LIN {X 0,Y 98.445,Z 539.877,A -85,B 0,C 180,E1 -26554.094,E2 -26554.094} C_VEL
LIN {X 0,Y 100.057,Z 537.535,A -85,B 0,C 180,E1 -26562.164,E2 -26562.164} C_VEL
LIN {X 0,Y 102.288,Z 534.743,A -85,B 0,C 180,E1 -26568.01,E2 -26568.01} C_VEL
LIN {X 0,Y 105.398,Z 531.036,A -85,B 0,C 180,E1 -26573.583,E2 -26573.583} C_VEL
LIN {X 0,Y 109.416,Z 526.315,A -85,B 0,C 180,E1 -26578.798,E2 -26578.798} C_VEL
LIN {X 0,Y 115.169,Z 519.342,A -85,B 0,C 180,E1 -26584.364,E2 -26584.364} C_VEL
LIN {X 0,Y 120.723,Z 511.905,A -85,B 0,C 180,E1 -26588.741,E2 -26588.741} C_VEL
LIN {X 0,Y 127.011,Z 502.792,A -85,B 0,C 180,E1 -26592.674,E2 -26592.674} C_VEL
LIN {X 0,Y 132.642,Z 493.502,A -85,B 0,C 180,E1 -26595.666,E2 -26595.666} C_VEL
LIN {X 0,Y 137.859,Z 483.367,A -85,B 0,C 180,E1 -26598.207,E2 -26598.207} C_VEL
LIN {X 0,Y 142.816,Z 472.376,A -85,B 0,C 180,E1 -26600.227,E2 -26600.227} C_VEL
LIN {X 0,Y 147.276,Z 460.103,A -85,B 0,C 180,E1 -26601.94,E2 -26601.94} C_VEL
LIN {X 0,Y 151.028,Z 446.667,A -85,B 0,C 180,E1 -26603.297,E2 -26603.297} C_VEL
LIN {X 0,Y 153.636,Z 433.846,A -85,B 0,C 180,E1 -26604.14,E2 -26604.14} C_VEL
LIN {X 0,Y 155.312,Z 419.503,A -85,B 0,C 180,E1 -26604.738,E2 -26604.738} C_VEL
LIN {X 0,Y 158.37,Z 382.753,A -85,B 0,C 180,E1 -26606.002,E2 -26606.002} C_VEL
LIN {X 0,Y 155.054,Z 373.648,A -85,B 0,C 180,E1 -26608.871,E2 -26608.871} C_VEL
LIN {X 0,Y 151.004,Z 364.193,A -85,B 0,C 180,E1 -26612.816,E2 -26612.816} C_VEL
LIN {X 0,Y 148.386,Z 358.823,A -85,B 0,C 180,E1 -26615.763,E2 -26615.763} C_VEL
LIN {X 0,Y 146.643,Z 355.474,A -85,B 0,C 180,E1 -26617.992,E2 -26617.992} C_VEL
LIN {X 0,Y 144.423,Z 351.265,A -85,B 0,C 180,E1 -26621.329,E2 -26621.329} C_VEL
LIN {X 0,Y 141.659,Z 346.333,A -85,B 0,C 180,E1 -26626.943,E2 -26626.943} C_VEL
LIN {X 0,Y 139.867,Z 343.216,A -85,B 0,C 180,E1 -26633.833,E2 -26633.833} C_VEL
LIN {X 0,Y 139.693,Z 342.139,A -85,B 0,C 180,E1 -26638.558,E2 -26638.558} C_VEL
LIN {X 0,Y 139.869,Z 342.535,A -85,B 0,C 180,E1 -26641.079,E2 -26641.079} C_VEL
LIN {X 0,Y 141.875,Z 345.546,A -85,B 0,C 180,E1 -26648.747,E2 -26648.747} C_VEL
LIN {X 0,Y 145.014,Z 350.889,A -85,B 0,C 180,E1 -26654.829,E2 -26654.829} C_VEL
LIN {X 0,Y 147.601,Z 355.381,A -85,B 0,C 180,E1 -26658.449,E2 -26658.449} C_VEL
LIN {X 0,Y 150.224,Z 360.312,A -85,B 0,C 180,E1 -26661.527,E2 -26661.527} C_VEL
LIN {X 0,Y 153.271,Z 366.548,A -85,B 0,C 180,E1 -26664.643,E2 -26664.643} C_VEL
LIN {X 0,Y 156.605,Z 374.178,A -85,B 0,C 180,E1 -26667.662,E2 -26667.662} C_VEL
LIN {X 0,Y 158.852,Z 380.327,A -85,B 0,C 180,E1 -26669.571,E2 -26669.571} C_VEL
LIN {X 0,Y 154.248,Z 429.807,A -85,B 0,C 180,E1 -26671.258,E2 -26671.258} C_VEL
LIN {X 0,Y 151.821,Z 443.678,A -85,B 0,C 180,E1 -26672.049,E2 -26672.049} C_VEL
LIN {X 0,Y 148.088,Z 457.884,A -85,B 0,C 180,E1 -26673.235,E2 -26673.235} C_VEL
LIN {X 0,Y 144.21,Z 469.529,A -85,B 0,C 180,E1 -26674.676,E2 -26674.676} C_VEL
LIN {X 0,Y 139.076,Z 481.819,A -85,B 0,C 180,E1 -26676.659,E2 -26676.659} C_VEL
LIN {X 0,Y 133.918,Z 492.462,A -85,B 0,C 180,E1 -26679.031,E2 -26679.031} C_VEL
LIN {X 0,Y 127.84,Z 503.024,A -85,B 0,C 180,E1 -26682.085,E2 -26682.085} C_VEL
LIN {X 0,Y 121.244,Z 512.968,A -85,B 0,C 180,E1 -26685.927,E2 -26685.927} C_VEL
LIN {X 0,Y 115.415,Z 521.126,A -85,B 0,C 180,E1 -26690.256,E2 -26690.256} C_VEL
LIN {X 0,Y 110.286,Z 527.828,A -85,B 0,C 180,E1 -26695.004,E2 -26695.004} C_VEL
LIN {X 0,Y 106.098,Z 533.312,A -85,B 0,C 180,E1 -26700.212,E2 -26700.212} C_VEL
LIN {X 0,Y 102.683,Z 537.722,A -85,B 0,C 180,E1 -26705.754,E2 -26705.754} C_VEL
LIN {X 0,Y 99.505,Z 542.086,A -85,B 0,C 180,E1 -26713.59,E2 -26713.59} C_VEL
LIN {X 0,Y 98.09,Z 544.903,A -85,B 0,C 180,E1 -26721.762,E2 -26721.762} C_VEL
LIN {X 0,Y 97.925,Z 545.745,A -85,B 0,C 180,E1 -26725.885,E2 -26725.885} C_VEL
LIN {X 0,Y 98.071,Z 546.205,A -85,B 0,C 180,E1 -26730,E2 -26730} C_VEL
LIN {X 0,Y 97.935,Z 546.283,A -85,B 0,C 180,E1 -26734.115,E2 -26734.115} C_VEL
LIN {X 0,Y 98.656,Z 545.36,A -85,B 0,C 180,E1 -26742.34,E2 -26742.34} C_VEL
LIN {X 0,Y 100.917,Z 542.994,A -85,B 0,C 180,E1 -26750.377,E2 -26750.377} C_VEL
LIN {X 0,Y 103.898,Z 540.216,A -85,B 0,C 180,E1 -26756.083,E2 -26756.083} C_VEL
LIN {X 0,Y 108.683,Z 535.456,A -85,B 0,C 180,E1 -26762.793,E2 -26762.793} C_VEL
LIN {X 0,Y 113.953,Z 530.064,A -85,B 0,C 180,E1 -26768.078,E2 -26768.078} C_VEL
LIN {X 0,Y 120.709,Z 522.772,A -85,B 0,C 180,E1 -26773.165,E2 -26773.165} C_VEL
LIN {X 0,Y 127.182,Z 515.033,A -85,B 0,C 180,E1 -26777.069,E2 -26777.069} C_VEL
LIN {X 0,Y 134.163,Z 505.579,A -85,B 0,C 180,E1 -26780.593,E2 -26780.593} C_VEL
LIN {X 0,Y 138.497,Z 498.922,A -85,B 0,C 180,E1 -26782.545,E2 -26782.545} C_VEL
LIN {X 0,Y 140.818,Z 494.528,A -85,B 0,C 180,E1 -26783.862,E2 -26783.862} C_VEL
LIN {X 0,Y 143.313,Z 487.207,A -85,B 0,C 180,E1 -26786.378,E2 -26786.378} C_VEL
LIN {X 0,Y 145.665,Z 479.481,A -85,B 0,C 180,E1 -26788.651,E2 -26788.651} C_VEL
LIN {X 0,Y 147.649,Z 474.457,A -85,B 0,C 180,E1 -26789.573,E2 -26789.573} C_VEL
LIN {X 0,Y 151.923,Z 464.012,A -85,B 0,C 180,E1 -26790.827,E2 -26790.827} C_VEL
LIN {X 0,Y 156.228,Z 450.743,A -85,B 0,C 180,E1 -26791.985,E2 -26791.985} C_VEL
LIN {X 0,Y 159.545,Z 436.77,A -85,B 0,C 180,E1 -26792.801,E2 -26792.801} C_VEL
LIN {X 0,Y 161.561,Z 422.766,A -85,B 0,C 180,E1 -26793.348,E2 -26793.348} C_VEL
LIN {X 0,Y 164.54,Z 391.448,A -85,B 0,C 180,E1 -26794.328,E2 -26794.328} C_VEL
LIN {X 0,Y 161.223,Z 382.87,A -85,B 0,C 180,E1 -26797.832,E2 -26797.832} C_VEL
LIN {X 0,Y 158.331,Z 376.36,A -85,B 0,C 180,E1 -26801.396,E2 -26801.396} C_VEL
LIN {X 0,Y 156.515,Z 372.65,A -85,B 0,C 180,E1 -26804.041,E2 -26804.041} C_VEL
LIN {X 0,Y 154.7,Z 369.18,A -85,B 0,C 180,E1 -26807.205,E2 -26807.205} C_VEL
LIN {X 0,Y 152.882,Z 365.51,A -85,B 0,C 180,E1 -26811.596,E2 -26811.596} C_VEL
LIN {X 0,Y 151.763,Z 363.688,A -85,B 0,C 180,E1 -26816.018,E2 -26816.018} C_VEL
LIN {X 0,Y 151.454,Z 362.725,A -85,B 0,C 180,E1 -26820.001,E2 -26820.001} C_VEL
LIN {X 0,Y 151.968,Z 364.564,A -85,B 0,C 180,E1 -26825.974,E2 -26825.974} C_VEL
LIN {X 0,Y 153.384,Z 367.616,A -85,B 0,C 180,E1 -26830.729,E2 -26830.729} C_VEL
LIN {X 0,Y 155.623,Z 372.465,A -85,B 0,C 180,E1 -26835.387,E2 -26835.387} C_VEL
LIN {X 0,Y 157.722,Z 377.127,A -85,B 0,C 180,E1 -26838.663,E2 -26838.663} C_VEL
LIN {X 0,Y 160.038,Z 382.681,A -85,B 0,C 180,E1 -26841.683,E2 -26841.683} C_VEL
LIN {X 0,Y 163.374,Z 391.759,A -85,B 0,C 180,E1 -26845.411,E2 -26845.411} C_VEL
LIN {X 0,Y 164.211,Z 394.346,A -85,B 0,C 180,E1 -26846.277,E2 -26846.277} C_VEL
LIN {X 0,Y 160.771,Z 429.208,A -85,B 0,C 180,E1 -26847.356,E2 -26847.356} C_VEL
LIN {X 0,Y 158.038,Z 443.429,A -85,B 0,C 180,E1 -26848.062,E2 -26848.062} C_VEL
LIN {X 0,Y 154.281,Z 456.733,A -85,B 0,C 180,E1 -26849.069,E2 -26849.069} C_VEL
LIN {X 0,Y 149.779,Z 468.983,A -85,B 0,C 180,E1 -26850.437,E2 -26850.437} C_VEL
LIN {X 0,Y 144.308,Z 480.728,A -85,B 0,C 180,E1 -26852.202,E2 -26852.202} C_VEL
LIN {X 0,Y 138.053,Z 491.906,A -85,B 0,C 180,E1 -26854.496,E2 -26854.496} C_VEL
LIN {X 0,Y 131.861,Z 501.111,A -85,B 0,C 180,E1 -26856.921,E2 -26856.921} C_VEL
LIN {X 0,Y 124.436,Z 510.659,A -85,B 0,C 180,E1 -26860.319,E2 -26860.319} C_VEL
LIN {X 0,Y 117.571,Z 518.415,A -85,B 0,C 180,E1 -26864.167,E2 -26864.167} C_VEL
LIN {X 0,Y 111.241,Z 524.729,A -85,B 0,C 180,E1 -26868.443,E2 -26868.443} C_VEL
LIN {X 0,Y 105.741,Z 529.827,A -85,B 0,C 180,E1 -26873.261,E2 -26873.261} C_VEL
LIN {X 0,Y 100.987,Z 533.857,A -85,B 0,C 180,E1 -26878.537,E2 -26878.537} C_VEL
LIN {X 0,Y 96.967,Z 536.935,A -85,B 0,C 180,E1 -26884.223,E2 -26884.223} C_VEL
LIN {X 0,Y 93.331,Z 539.678,A -85,B 0,C 180,E1 -26892.47,E2 -26892.47} C_VEL
LIN {X 0,Y 91.373,Z 540.926,A -85,B 0,C 180,E1 -26901.151,E2 -26901.151} C_VEL
LIN {X 0,Y 91.052,Z 540.719,A -85,B 0,C 180,E1 -26910,E2 -26910} C_VEL
LIN {X 0,Y 91.387,Z 540.09,A -85,B 0,C 180,E1 -26914.41,E2 -26914.41} C_VEL
LIN {X 0,Y 93.142,Z 537.76,A -85,B 0,C 180,E1 -26923.083,E2 -26923.083} C_VEL
LIN {X 0,Y 95.566,Z 534.981,A -85,B 0,C 180,E1 -26929.325,E2 -26929.325} C_VEL
LIN {X 0,Y 98.954,Z 531.289,A -85,B 0,C 180,E1 -26935.222,E2 -26935.222} C_VEL
LIN {X 0,Y 103.263,Z 526.585,A -85,B 0,C 180,E1 -26940.693,E2 -26940.693} C_VEL
LIN {X 0,Y 109.397,Z 519.632,A -85,B 0,C 180,E1 -26946.458,E2 -26946.458} C_VEL
LIN {X 0,Y 115.273,Z 512.221,A -85,B 0,C 180,E1 -26950.95,E2 -26950.95} C_VEL
LIN {X 0,Y 121.91,Z 503.144,A -85,B 0,C 180,E1 -26954.926,E2 -26954.926} C_VEL
LIN {X 0,Y 126.607,Z 495.855,A -85,B 0,C 180,E1 -26957.349,E2 -26957.349} C_VEL
LIN {X 0,Y 132.616,Z 485.046,A -85,B 0,C 180,E1 -26960.211,E2 -26960.211} C_VEL
LIN {X 0,Y 138.024,Z 473.823,A -85,B 0,C 180,E1 -26962.335,E2 -26962.335} C_VEL
LIN {X 0,Y 142.375,Z 462.739,A -85,B 0,C 180,E1 -26963.93,E2 -26963.93} C_VEL
LIN {X 0,Y 146.275,Z 449.923,A -85,B 0,C 180,E1 -26965.307,E2 -26965.307} C_VEL
LIN {X 0,Y 149.398,Z 436.136,A -85,B 0,C 180,E1 -26966.274,E2 -26966.274} C_VEL
LIN {X 0,Y 151.259,Z 422.842,A -85,B 0,C 180,E1 -26966.869,E2 -26966.869} C_VEL
LIN {X 0,Y 154.537,Z 385.412,A -85,B 0,C 180,E1 -26968.135,E2 -26968.135} C_VEL
LIN {X 0,Y 151.217,Z 376.194,A -85,B 0,C 180,E1 -26971.37,E2 -26971.37} C_VEL
LIN {X 0,Y 147.848,Z 368.107,A -85,B 0,C 180,E1 -26975.115,E2 -26975.115} C_VEL
LIN {X 0,Y 145.186,Z 362.309,A -85,B 0,C 180,E1 -26978.625,E2 -26978.625} C_VEL
LIN {X 0,Y 142.907,Z 357.801,A -85,B 0,C 180,E1 -26982.283,E2 -26982.283} C_VEL
LIN {X 0,Y 140.493,Z 353.11,A -85,B 0,C 180,E1 -26987.651,E2 -26987.651} C_VEL
LIN {X 0,Y 138.91,Z 350.107,A -85,B 0,C 180,E1 -26994.566,E2 -26994.566} C_VEL
LIN {X 0,Y 138.826,Z 349.201,A -85,B 0,C 180,E1 -26998.549,E2 -26998.549} C_VEL
LIN {X 0,Y 138.996,Z 349.636,A -85,B 0,C 180,E1 -27001.085,E2 -27001.085} C_VEL
LIN {X 0,Y 140.772,Z 352.508,A -85,B 0,C 180,E1 -27008.251,E2 -27008.251} C_VEL
LIN {X 0,Y 143.481,Z 357.418,A -85,B 0,C 180,E1 -27013.904,E2 -27013.904} C_VEL
LIN {X 0,Y 145.753,Z 361.641,A -85,B 0,C 180,E1 -27017.358,E2 -27017.358} C_VEL
LIN {X 0,Y 148.347,Z 366.881,A -85,B 0,C 180,E1 -27020.653,E2 -27020.653} C_VEL
LIN {X 0,Y 151.329,Z 373.477,A -85,B 0,C 180,E1 -27023.908,E2 -27023.908} C_VEL
LIN {X 0,Y 154.651,Z 381.947,A -85,B 0,C 180,E1 -27027.119,E2 -27027.119} C_VEL
LIN {X 0,Y 154.977,Z 382.874,A -85,B 0,C 180,E1 -27027.419,E2 -27027.419} C_VEL
LIN {X 0,Y 150.424,Z 430.008,A -85,B 0,C 180,E1 -27029.013,E2 -27029.013} C_VEL
LIN {X 0,Y 147.841,Z 444.116,A -85,B 0,C 180,E1 -27029.807,E2 -27029.807} C_VEL
LIN {X 0,Y 144.302,Z 457.156,A -85,B 0,C 180,E1 -27030.865,E2 -27030.865} C_VEL
LIN {X 0,Y 140.279,Z 468.942,A -85,B 0,C 180,E1 -27032.283,E2 -27032.283} C_VEL
LIN {X 0,Y 134.925,Z 481.329,A -85,B 0,C 180,E1 -27034.22,E2 -27034.22} C_VEL
LIN {X 0,Y 128.968,Z 493.038,A -85,B 0,C 180,E1 -27036.828,E2 -27036.828} C_VEL
LIN {X 0,Y 123.148,Z 502.661,A -85,B 0,C 180,E1 -27039.608,E2 -27039.608} C_VEL
LIN {X 0,Y 116.234,Z 512.64,A -85,B 0,C 180,E1 -27043.485,E2 -27043.485} C_VEL
LIN {X 0,Y 110.002,Z 520.823,A -85,B 0,C 180,E1 -27047.869,E2 -27047.869} C_VEL
LIN {X 0,Y 104.503,Z 527.547,A -85,B 0,C 180,E1 -27052.753,E2 -27052.753} C_VEL
LIN {X 0,Y 99.89,Z 533.093,A -85,B 0,C 180,E1 -27058.217,E2 -27058.217} C_VEL
LIN {X 0,Y 95.158,Z 538.74,A -85,B 0,C 180,E1 -27066.034,E2 -27066.034} C_VEL
LIN {X 0,Y 92.674,Z 541.853,A -85,B 0,C 180,E1 -27072.342,E2 -27072.342} C_VEL
LIN {X 0,Y 91.056,Z 544.683,A -85,B 0,C 180,E1 -27081.12,E2 -27081.12} C_VEL
LIN {X 0,Y 90.824,Z 545.535,A -85,B 0,C 180,E1 -27085.562,E2 -27085.562} C_VEL
LIN {X 0,Y 90.969,Z 546.003,A -85,B 0,C 180,E1 -27090,E2 -27090} C_VEL
LIN {X 0,Y 90.861,Z 546.087,A -85,B 0,C 180,E1 -27094.436,E2 -27094.436} C_VEL
LIN {X 0,Y 91.684,Z 545.173,A -85,B 0,C 180,E1 -27103.295,E2 -27103.295} C_VEL
LIN {X 0,Y 94.253,Z 542.817,A -85,B 0,C 180,E1 -27111.89,E2 -27111.89} C_VEL
LIN {X 0,Y 97.518,Z 540.049,A -85,B 0,C 180,E1 -27117.933,E2 -27117.933} C_VEL
LIN {X 0,Y 102.319,Z 535.68,A -85,B 0,C 180,E1 -27124.49,E2 -27124.49} C_VEL
LIN {X 0,Y 108.424,Z 529.917,A -85,B 0,C 180,E1 -27130.405,E2 -27130.405} C_VEL
LIN {X 0,Y 115.578,Z 522.633,A -85,B 0,C 180,E1 -27135.6,E2 -27135.6} C_VEL
LIN {X 0,Y 122.433,Z 514.904,A -85,B 0,C 180,E1 -27139.515,E2 -27139.515} C_VEL
LIN {X 0,Y 129.75,Z 505.459,A -85,B 0,C 180,E1 -27143.028,E2 -27143.028} C_VEL
LIN {X 0,Y 136.785,Z 494.847,A -85,B 0,C 180,E1 -27145.944,E2 -27145.944} C_VEL
LIN {X 0,Y 143.528,Z 482.98,A -85,B 0,C 180,E1 -27148.296,E2 -27148.296} C_VEL
LIN {X 0,Y 147.649,Z 474.457,A -85,B 0,C 180,E1 -27149.573,E2 -27149.573} C_VEL
LIN {X 0,Y 149.552,Z 469.346,A -85,B 0,C 180,E1 -27150.423,E2 -27150.423} C_VEL
LIN {X 0,Y 151.378,Z 460.868,A -85,B 0,C 180,E1 -27152.289,E2 -27152.289} C_VEL
LIN {X 0,Y 152.891,Z 452.178,A -85,B 0,C 180,E1 -27153.992,E2 -27153.992} C_VEL
LIN {X 0,Y 154.136,Z 446.643,A -85,B 0,C 180,E1 -27154.595,E2 -27154.595} C_VEL
LIN {X 0,Y 157.082,Z 432.911,A -85,B 0,C 180,E1 -27155.283,E2 -27155.283} C_VEL
LIN {X 0,Y 159.335,Z 414.404,A -85,B 0,C 180,E1 -27155.864,E2 -27155.864} C_VEL
LIN {X 0,Y 161.221,Z 394.644,A -85,B 0,C 180,E1 -27156.512,E2 -27156.512} C_VEL
LIN {X 0,Y 158.447,Z 387.195,A -85,B 0,C 180,E1 -27159.831,E2 -27159.831} C_VEL
LIN {X 0,Y 156.284,Z 381.996,A -85,B 0,C 180,E1 -27162.855,E2 -27162.855} C_VEL
LIN {X 0,Y 154.65,Z 378.477,A -85,B 0,C 180,E1 -27165.527,E2 -27165.527} C_VEL
LIN {X 0,Y 153.338,Z 375.711,A -85,B 0,C 180,E1 -27168.098,E2 -27168.098} C_VEL
LIN {X 0,Y 151.747,Z 372.291,A -85,B 0,C 180,E1 -27172.349,E2 -27172.349} C_VEL
LIN {X 0,Y 150.896,Z 370.762,A -85,B 0,C 180,E1 -27175.995,E2 -27175.995} C_VEL
LIN {X 0,Y 150.587,Z 369.788,A -85,B 0,C 180,E1 -27180.001,E2 -27180.001} C_VEL
LIN {X 0,Y 151.004,Z 371.517,A -85,B 0,C 180,E1 -27185.509,E2 -27185.509} C_VEL
LIN {X 0,Y 152.203,Z 374.306,A -85,B 0,C 180,E1 -27189.972,E2 -27189.972} C_VEL
LIN {X 0,Y 154.186,Z 379.039,A -85,B 0,C 180,E1 -27194.52,E2 -27194.52} C_VEL
LIN {X 0,Y 155.977,Z 383.346,A -85,B 0,C 180,E1 -27197.58,E2 -27197.58} C_VEL
LIN {X 0,Y 158.065,Z 388.862,A -85,B 0,C 180,E1 -27200.581,E2 -27200.581} C_VEL
LIN {X 0,Y 160.793,Z 396.887,A -85,B 0,C 180,E1 -27203.935,E2 -27203.935} C_VEL
LIN {X 0,Y 160.927,Z 397.28,A -85,B 0,C 180,E1 -27204.085,E2 -27204.085} C_VEL
LIN {X 0,Y 157.648,Z 429.259,A -85,B 0,C 180,E1 -27205.057,E2 -27205.057} C_VEL
LIN {X 0,Y 155.029,Z 442.78,A -85,B 0,C 180,E1 -27205.712,E2 -27205.712} C_VEL
LIN {X 0,Y 151.334,Z 455.704,A -85,B 0,C 180,E1 -27206.625,E2 -27206.625} C_VEL
LIN {X 0,Y 147.017,Z 467.353,A -85,B 0,C 180,E1 -27207.827,E2 -27207.827} C_VEL
LIN {X 0,Y 141.346,Z 479.535,A -85,B 0,C 180,E1 -27209.528,E2 -27209.528} C_VEL
LIN {X 0,Y 134.935,Z 490.768,A -85,B 0,C 180,E1 -27211.699,E2 -27211.699} C_VEL
LIN {X 0,Y 127.726,Z 501.224,A -85,B 0,C 180,E1 -27214.376,E2 -27214.376} C_VEL
LIN {X 0,Y 119.954,Z 510.781,A -85,B 0,C 180,E1 -27217.727,E2 -27217.727} C_VEL
LIN {X 0,Y 112.723,Z 518.547,A -85,B 0,C 180,E1 -27221.569,E2 -27221.569} C_VEL
LIN {X 0,Y 106.025,Z 524.87,A -85,B 0,C 180,E1 -27225.893,E2 -27225.893} C_VEL
LIN {X 0,Y 100.095,Z 529.977,A -85,B 0,C 180,E1 -27230.809,E2 -27230.809} C_VEL
LIN {X 0,Y 94.98,Z 534.016,A -85,B 0,C 180,E1 -27236.293,E2 -27236.293} C_VEL
LIN {X 0,Y 90.607,Z 537.104,A -85,B 0,C 180,E1 -27242.265,E2 -27242.265} C_VEL
LIN {X 0,Y 86.578,Z 539.858,A -85,B 0,C 180,E1 -27251.053,E2 -27251.053} C_VEL
LIN {X 0,Y 84.368,Z 541.122,A -85,B 0,C 180,E1 -27260.41,E2 -27260.41} C_VEL
LIN {X 0,Y 83.952,Z 540.927,A -85,B 0,C 180,E1 -27270,E2 -27270} C_VEL
LIN {X 0,Y 84.319,Z 540.303,A -85,B 0,C 180,E1 -27274.781,E2 -27274.781} C_VEL
LIN {X 0,Y 86.245,Z 537.985,A -85,B 0,C 180,E1 -27284.15,E2 -27284.15} C_VEL
LIN {X 0,Y 88.892,Z 535.22,A -85,B 0,C 180,E1 -27290.841,E2 -27290.841} C_VEL
LIN {X 0,Y 92.579,Z 531.542,A -85,B 0,C 180,E1 -27297.095,E2 -27297.095} C_VEL
LIN {X 0,Y 97.24,Z 526.855,A -85,B 0,C 180,E1 -27302.823,E2 -27302.823} C_VEL
LIN {X 0,Y 103.787,Z 519.923,A -85,B 0,C 180,E1 -27308.782,E2 -27308.782} C_VEL
LIN {X 0,Y 110.016,Z 512.537,A -85,B 0,C 180,E1 -27313.371,E2 -27313.371} C_VEL
LIN {X 0,Y 117.012,Z 503.49,A -85,B 0,C 180,E1 -27317.37,E2 -27317.37} C_VEL
LIN {X 0,Y 121.917,Z 496.239,A -85,B 0,C 180,E1 -27319.8,E2 -27319.8} C_VEL
LIN {X 0,Y 128.207,Z 485.478,A -85,B 0,C 180,E1 -27322.64,E2 -27322.64} C_VEL
LIN {X 0,Y 133.331,Z 475.365,A -85,B 0,C 180,E1 -27324.561,E2 -27324.561} C_VEL
LIN {X 0,Y 138.328,Z 463.371,A -85,B 0,C 180,E1 -27326.299,E2 -27326.299} C_VEL
LIN {X 0,Y 142.37,Z 450.796,A -85,B 0,C 180,E1 -27327.638,E2 -27327.638} C_VEL
LIN {X 0,Y 145.53,Z 437.606,A -85,B 0,C 180,E1 -27328.572,E2 -27328.572} C_VEL
LIN {X 0,Y 147.65,Z 423.589,A -85,B 0,C 180,E1 -27329.207,E2 -27329.207} C_VEL
LIN {X 0,Y 150.893,Z 388.267,A -85,B 0,C 180,E1 -27330.381,E2 -27330.381} C_VEL
LIN {X 0,Y 148.35,Z 380.843,A -85,B 0,C 180,E1 -27333.173,E2 -27333.173} C_VEL
LIN {X 0,Y 145.424,Z 373.222,A -85,B 0,C 180,E1 -27336.831,E2 -27336.831} C_VEL
LIN {X 0,Y 143.128,Z 368.019,A -85,B 0,C 180,E1 -27340.211,E2 -27340.211} C_VEL
LIN {X 0,Y 141.406,Z 364.287,A -85,B 0,C 180,E1 -27343.307,E2 -27343.307} C_VEL
LIN {X 0,Y 139.349,Z 359.916,A -85,B 0,C 180,E1 -27348.36,E2 -27348.36} C_VEL
LIN {X 0,Y 137.98,Z 356.979,A -85,B 0,C 180,E1 -27355.284,E2 -27355.284} C_VEL
LIN {X 0,Y 137.92,Z 356.533,A -85,B 0,C 180,E1 -27357.078,E2 -27357.078} C_VEL
LIN {X 0,Y 138.06,Z 356.51,A -85,B 0,C 180,E1 -27360.364,E2 -27360.364} C_VEL
LIN {X 0,Y 139.629,Z 359.345,A -85,B 0,C 180,E1 -27367.591,E2 -27367.591} C_VEL
LIN {X 0,Y 142.126,Z 364.234,A -85,B 0,C 180,E1 -27373.22,E2 -27373.22} C_VEL
LIN {X 0,Y 144.103,Z 368.243,A -85,B 0,C 180,E1 -27376.467,E2 -27376.467} C_VEL
LIN {X 0,Y 146.651,Z 373.729,A -85,B 0,C 180,E1 -27379.925,E2 -27379.925} C_VEL
LIN {X 0,Y 149.624,Z 381.135,A -85,B 0,C 180,E1 -27383.404,E2 -27383.404} C_VEL
LIN {X 0,Y 151.295,Z 385.731,A -85,B 0,C 180,E1 -27385.167,E2 -27385.167} C_VEL
LIN {X 0,Y 146.794,Z 430.509,A -85,B 0,C 180,E1 -27386.667,E2 -27386.667} C_VEL
LIN {X 0,Y 144.14,Z 444.415,A -85,B 0,C 180,E1 -27387.442,E2 -27387.442} C_VEL
LIN {X 0,Y 140.421,Z 457.561,A -85,B 0,C 180,E1 -27388.481,E2 -27388.481} C_VEL
LIN {X 0,Y 135.906,Z 470.127,A -85,B 0,C 180,E1 -27389.985,E2 -27389.985} C_VEL
LIN {X 0,Y 130.362,Z 482.213,A -85,B 0,C 180,E1 -27391.888,E2 -27391.888} C_VEL
LIN {X 0,Y 124.242,Z 493.586,A -85,B 0,C 180,E1 -27394.448,E2 -27394.448} C_VEL
LIN {X 0,Y 117.507,Z 504.1,A -85,B 0,C 180,E1 -27397.584,E2 -27397.584} C_VEL
LIN {X 0,Y 110.262,Z 513.811,A -85,B 0,C 180,E1 -27401.503,E2 -27401.503} C_VEL
LIN {X 0,Y 103.77,Z 521.767,A -85,B 0,C 180,E1 -27406.038,E2 -27406.038} C_VEL
LIN {X 0,Y 97.107,Z 529.248,A -85,B 0,C 180,E1 -27412.036,E2 -27412.036} C_VEL
LIN {X 0,Y 92.466,Z 534.409,A -85,B 0,C 180,E1 -27417.857,E2 -27417.857} C_VEL
LIN {X 0,Y 88.662,Z 538.493,A -85,B 0,C 180,E1 -27424.154,E2 -27424.154} C_VEL
LIN {X 0,Y 85.876,Z 541.62,A -85,B 0,C 180,E1 -27430.892,E2 -27430.892} C_VEL
LIN {X 0,Y 84.018,Z 544.464,A -85,B 0,C 180,E1 -27440.37,E2 -27440.37} C_VEL
LIN {X 0,Y 83.747,Z 545.325,A -85,B 0,C 180,E1 -27445.186,E2 -27445.186} C_VEL
LIN {X 0,Y 83.875,Z 545.802,A -85,B 0,C 180,E1 -27450,E2 -27450} C_VEL
LIN {X 0,Y 83.775,Z 545.89,A -85,B 0,C 180,E1 -27454.812,E2 -27454.812} C_VEL
LIN {X 0,Y 84.753,Z 544.987,A -85,B 0,C 180,E1 -27464.405,E2 -27464.405} C_VEL
LIN {X 0,Y 87.671,Z 542.641,A -85,B 0,C 180,E1 -27473.629,E2 -27473.629} C_VEL
LIN {X 0,Y 91.244,Z 539.883,A -85,B 0,C 180,E1 -27480.043,E2 -27480.043} C_VEL
LIN {X 0,Y 97.229,Z 534.929,A -85,B 0,C 180,E1 -27487.646,E2 -27487.646} C_VEL
LIN {X 0,Y 103.075,Z 529.77,A -85,B 0,C 180,E1 -27492.986,E2 -27492.986} C_VEL
LIN {X 0,Y 110.693,Z 522.496,A -85,B 0,C 180,E1 -27498.246,E2 -27498.246} C_VEL
LIN {X 0,Y 117.924,Z 514.775,A -85,B 0,C 180,E1 -27502.154,E2 -27502.154} C_VEL
LIN {X 0,Y 125.595,Z 505.34,A -85,B 0,C 180,E1 -27505.625,E2 -27505.625} C_VEL
LIN {X 0,Y 132.922,Z 494.734,A -85,B 0,C 180,E1 -27508.492,E2 -27508.492} C_VEL
LIN {X 0,Y 139.926,Z 482.871,A -85,B 0,C 180,E1 -27510.771,E2 -27510.771} C_VEL
LIN {X 0,Y 145.652,Z 471.059,A -85,B 0,C 180,E1 -27512.451,E2 -27512.451} C_VEL
LIN {X 0,Y 150.807,Z 457.754,A -85,B 0,C 180,E1 -27513.778,E2 -27513.778} C_VEL
LIN {X 0,Y 154.136,Z 446.643,A -85,B 0,C 180,E1 -27514.595,E2 -27514.595} C_VEL
LIN {X 0,Y 155.242,Z 441.025,A -85,B 0,C 180,E1 -27515.122,E2 -27515.122} C_VEL
LIN {X 0,Y 155.853,Z 431.841,A -85,B 0,C 180,E1 -27516.459,E2 -27516.459} C_VEL
LIN {X 0,Y 155.986,Z 422.547,A -85,B 0,C 180,E1 -27517.74,E2 -27517.74} C_VEL
LIN {X 0,Y 156.29,Z 416.752,A -85,B 0,C 180,E1 -27518.167,E2 -27518.167} C_VEL
LIN {X 0,Y 158.157,Z 398.049,A -85,B 0,C 180,E1 -27518.745,E2 -27518.745} C_VEL
LIN {X 0,Y 155.899,Z 391.587,A -85,B 0,C 180,E1 -27521.87,E2 -27521.87} C_VEL
LIN {X 0,Y 153.826,Z 386.293,A -85,B 0,C 180,E1 -27525.278,E2 -27525.278} C_VEL
LIN {X 0,Y 152.011,Z 382.264,A -85,B 0,C 180,E1 -27529.006,E2 -27529.006} C_VEL
LIN {X 0,Y 150.679,Z 379.133,A -85,B 0,C 180,E1 -27532.968,E2 -27532.968} C_VEL
LIN {X 0,Y 149.926,Z 377.679,A -85,B 0,C 180,E1 -27536.642,E2 -27536.642} C_VEL
LIN {X 0,Y 149.722,Z 376.829,A -85,B 0,C 180,E1 -27540.001,E2 -27540.001} C_VEL
LIN {X 0,Y 150.027,Z 378.341,A -85,B 0,C 180,E1 -27544.872,E2 -27544.872} C_VEL
LIN {X 0,Y 151.093,Z 381.191,A -85,B 0,C 180,E1 -27549.37,E2 -27549.37} C_VEL
LIN {X 0,Y 152.826,Z 385.696,A -85,B 0,C 180,E1 -27553.718,E2 -27553.718} C_VEL
LIN {X 0,Y 154.52,Z 390.184,A -85,B 0,C 180,E1 -27556.865,E2 -27556.865} C_VEL
LIN {X 0,Y 156.369,Z 395.675,A -85,B 0,C 180,E1 -27559.757,E2 -27559.757} C_VEL
LIN {X 0,Y 157.885,Z 400.655,A -85,B 0,C 180,E1 -27561.859,E2 -27561.859} C_VEL
LIN {X 0,Y 154.781,Z 429.411,A -85,B 0,C 180,E1 -27562.681,E2 -27562.681} C_VEL
LIN {X 0,Y 152.093,Z 442.894,A -85,B 0,C 180,E1 -27563.31,E2 -27563.31} C_VEL
LIN {X 0,Y 148.298,Z 455.806,A -85,B 0,C 180,E1 -27564.18,E2 -27564.18} C_VEL
LIN {X 0,Y 143.834,Z 467.452,A -85,B 0,C 180,E1 -27565.32,E2 -27565.32} C_VEL
LIN {X 0,Y 137.982,Z 479.636,A -85,B 0,C 180,E1 -27566.959,E2 -27566.959} C_VEL
LIN {X 0,Y 132.283,Z 489.398,A -85,B 0,C 180,E1 -27568.723,E2 -27568.723} C_VEL
LIN {X 0,Y 125.242,Z 499.563,A -85,B 0,C 180,E1 -27571.158,E2 -27571.158} C_VEL
LIN {X 0,Y 117.05,Z 509.425,A -85,B 0,C 180,E1 -27574.353,E2 -27574.353} C_VEL
LIN {X 0,Y 109.381,Z 517.459,A -85,B 0,C 180,E1 -27578.086,E2 -27578.086} C_VEL
LIN {X 0,Y 101.034,Z 525.012,A -85,B 0,C 180,E1 -27583.082,E2 -27583.082} C_VEL
LIN {X 0,Y 94.649,Z 530.127,A -85,B 0,C 180,E1 -27588.066,E2 -27588.066} C_VEL
LIN {X 0,Y 89.126,Z 534.176,A -85,B 0,C 180,E1 -27593.743,E2 -27593.743} C_VEL
LIN {X 0,Y 84.373,Z 537.273,A -85,B 0,C 180,E1 -27600.015,E2 -27600.015} C_VEL
LIN {X 0,Y 79.857,Z 540.039,A -85,B 0,C 180,E1 -27609.389,E2 -27609.389} C_VEL
LIN {X 0,Y 78.374,Z 540.869,A -85,B 0,C 180,E1 -27614.394,E2 -27614.394} C_VEL
LIN {X 0,Y 76.876,Z 541.402,A -85,B 0,C 180,E1 -27624.755,E2 -27624.755} C_VEL
LIN {X 0,Y 76.859,Z 541.134,A -85,B 0,C 180,E1 -27630,E2 -27630} C_VEL
LIN {X 0,Y 77.249,Z 540.516,A -85,B 0,C 180,E1 -27635.22,E2 -27635.22} C_VEL
LIN {X 0,Y 79.399,Z 538.209,A -85,B 0,C 180,E1 -27645.399,E2 -27645.399} C_VEL
LIN {X 0,Y 82.295,Z 535.458,A -85,B 0,C 180,E1 -27652.6,E2 -27652.6} C_VEL
LIN {X 0,Y 86.324,Z 531.796,A -85,B 0,C 180,E1 -27659.24,E2 -27659.24} C_VEL
LIN {X 0,Y 91.372,Z 527.125,A -85,B 0,C 180,E1 -27665.23,E2 -27665.23} C_VEL
LIN {X 0,Y 98.346,Z 520.214,A -85,B 0,C 180,E1 -27671.377,E2 -27671.377} C_VEL
LIN {X 0,Y 104.98,Z 512.851,A -85,B 0,C 180,E1 -27676.026,E2 -27676.026} C_VEL
LIN {X 0,Y 112.335,Z 503.834,A -85,B 0,C 180,E1 -27680.03,E2 -27680.03} C_VEL
LIN {X 0,Y 117.461,Z 496.623,A -85,B 0,C 180,E1 -27682.445,E2 -27682.445} C_VEL
LIN {X 0,Y 124.044,Z 485.911,A -85,B 0,C 180,E1 -27685.237,E2 -27685.237} C_VEL
LIN {X 0,Y 129.6,Z 475.381,A -85,B 0,C 180,E1 -27687.192,E2 -27687.192} C_VEL
LIN {X 0,Y 134.531,Z 463.973,A -85,B 0,C 180,E1 -27688.806,E2 -27688.806} C_VEL
LIN {X 0,Y 138.706,Z 451.671,A -85,B 0,C 180,E1 -27690.1,E2 -27690.1} C_VEL
LIN {X 0,Y 142.053,Z 438.325,A -85,B 0,C 180,E1 -27691.037,E2 -27691.037} C_VEL
LIN {X 0,Y 144.266,Z 424.743,A -85,B 0,C 180,E1 -27691.631,E2 -27691.631} C_VEL
LIN {X 0,Y 147.465,Z 392.041,A -85,B 0,C 180,E1 -27692.66,E2 -27692.66} C_VEL
LIN {X 0,Y 147.416,Z 390.899,A -85,B 0,C 180,E1 -27692.829,E2 -27692.829} C_VEL
LIN {X 0,Y 145.023,Z 383.651,A -85,B 0,C 180,E1 -27695.868,E2 -27695.868} C_VEL
LIN {X 0,Y 142.707,Z 377.322,A -85,B 0,C 180,E1 -27699.254,E2 -27699.254} C_VEL
LIN {X 0,Y 141.168,Z 373.694,A -85,B 0,C 180,E1 -27701.87,E2 -27701.87} C_VEL
LIN {X 0,Y 139.928,Z 370.726,A -85,B 0,C 180,E1 -27704.404,E2 -27704.404} C_VEL
LIN {X 0,Y 138.249,Z 366.755,A -85,B 0,C 180,E1 -27709.009,E2 -27709.009} C_VEL
LIN {X 0,Y 137.088,Z 363.973,A -85,B 0,C 180,E1 -27715.633,E2 -27715.633} C_VEL
LIN {X 0,Y 137.051,Z 363.612,A -85,B 0,C 180,E1 -27717.06,E2 -27717.06} C_VEL
LIN {X 0,Y 137.192,Z 363.57,A -85,B 0,C 180,E1 -27720.366,E2 -27720.366} C_VEL
LIN {X 0,Y 138.478,Z 366.151,A -85,B 0,C 180,E1 -27726.853,E2 -27726.853} C_VEL
LIN {X 0,Y 140.696,Z 370.861,A -85,B 0,C 180,E1 -27732.348,E2 -27732.348} C_VEL
LIN {X 0,Y 142.463,Z 374.773,A -85,B 0,C 180,E1 -27735.513,E2 -27735.513} C_VEL
LIN {X 0,Y 144.72,Z 380.122,A -85,B 0,C 180,E1 -27738.858,E2 -27738.858} C_VEL
LIN {X 0,Y 147.508,Z 387.714,A -85,B 0,C 180,E1 -27742.405,E2 -27742.405} C_VEL
LIN {X 0,Y 147.853,Z 388.738,A -85,B 0,C 180,E1 -27742.812,E2 -27742.812} C_VEL
LIN {X 0,Y 143.66,Z 429.593,A -85,B 0,C 180,E1 -27744.151,E2 -27744.151} C_VEL
LIN {X 0,Y 140.947,Z 443.642,A -85,B 0,C 180,E1 -27744.879,E2 -27744.879} C_VEL
LIN {X 0,Y 137.185,Z 456.837,A -85,B 0,C 180,E1 -27745.88,E2 -27745.88} C_VEL
LIN {X 0,Y 132.48,Z 469.538,A -85,B 0,C 180,E1 -27747.307,E2 -27747.307} C_VEL
LIN {X 0,Y 126.755,Z 481.75,A -85,B 0,C 180,E1 -27749.162,E2 -27749.162} C_VEL
LIN {X 0,Y 121.178,Z 491.791,A -85,B 0,C 180,E1 -27751.271,E2 -27751.271} C_VEL
LIN {X 0,Y 114.574,Z 501.938,A -85,B 0,C 180,E1 -27754.099,E2 -27754.099} C_VEL
LIN {X 0,Y 106.909,Z 511.984,A -85,B 0,C 180,E1 -27757.923,E2 -27757.923} C_VEL
LIN {X 0,Y 99.851,Z 520.219,A -85,B 0,C 180,E1 -27762.352,E2 -27762.352} C_VEL
LIN {X 0,Y 93.509,Z 526.986,A -85,B 0,C 180,E1 -27767.436,E2 -27767.436} C_VEL
LIN {X 0,Y 88.049,Z 532.512,A -85,B 0,C 180,E1 -27773.21,E2 -27773.21} C_VEL
LIN {X 0,Y 83.555,Z 536.984,A -85,B 0,C 180,E1 -27779.691,E2 -27779.691} C_VEL
LIN {X 0,Y 79.147,Z 541.388,A -85,B 0,C 180,E1 -27789.196,E2 -27789.196} C_VEL
LIN {X 0,Y 76.986,Z 544.244,A -85,B 0,C 180,E1 -27799.481,E2 -27799.481} C_VEL
LIN {X 0,Y 76.649,Z 545.113,A -85,B 0,C 180,E1 -27804.74,E2 -27804.74} C_VEL
LIN {X 0,Y 76.772,Z 545.6,A -85,B 0,C 180,E1 -27810,E2 -27810} C_VEL
LIN {X 0,Y 76.676,Z 545.693,A -85,B 0,C 180,E1 -27815.259,E2 -27815.259} C_VEL
LIN {X 0,Y 77.868,Z 544.8,A -85,B 0,C 180,E1 -27825.71,E2 -27825.71} C_VEL
LIN {X 0,Y 81.188,Z 542.465,A -85,B 0,C 180,E1 -27835.647,E2 -27835.647} C_VEL
LIN {X 0,Y 86.672,Z 538.63,A -85,B 0,C 180,E1 -27844.583,E2 -27844.583} C_VEL
LIN {X 0,Y 91.862,Z 534.628,A -85,B 0,C 180,E1 -27850.564,E2 -27850.564} C_VEL
LIN {X 0,Y 97.969,Z 529.623,A -85,B 0,C 180,E1 -27855.837,E2 -27855.837} C_VEL
LIN {X 0,Y 106.058,Z 522.358,A -85,B 0,C 180,E1 -27861.133,E2 -27861.133} C_VEL
LIN {X 0,Y 113.694,Z 514.646,A -85,B 0,C 180,E1 -27864.988,E2 -27864.988} C_VEL
LIN {X 0,Y 121.717,Z 505.22,A -85,B 0,C 180,E1 -27868.393,E2 -27868.393} C_VEL
LIN {X 0,Y 129.341,Z 494.62,A -85,B 0,C 180,E1 -27871.184,E2 -27871.184} C_VEL
LIN {X 0,Y 136.601,Z 482.762,A -85,B 0,C 180,E1 -27873.369,E2 -27873.369} C_VEL
LIN {X 0,Y 142.502,Z 470.951,A -85,B 0,C 180,E1 -27874.987,E2 -27874.987} C_VEL
LIN {X 0,Y 147.804,Z 457.639,A -85,B 0,C 180,E1 -27876.25,E2 -27876.25} C_VEL
LIN {X 0,Y 152.008,Z 443.441,A -85,B 0,C 180,E1 -27877.189,E2 -27877.189} C_VEL
LIN {X 0,Y 154.81,Z 429.344,A -85,B 0,C 180,E1 -27877.813,E2 -27877.813} C_VEL
LIN {X 0,Y 156.29,Z 416.752,A -85,B 0,C 180,E1 -27878.167,E2 -27878.167} C_VEL
LIN {X 0,Y 156.477,Z 412.785,A -85,B 0,C 180,E1 -27878.482,E2 -27878.482} C_VEL
LIN {X 0,Y 156.341,Z 409.038,A -85,B 0,C 180,E1 -27879.074,E2 -27879.074} C_VEL
LIN {X 0,Y 155.794,Z 404.501,A -85,B 0,C 180,E1 -27880.192,E2 -27880.192} C_VEL
LIN {X 0,Y 154.966,Z 400.579,A -85,B 0,C 180,E1 -27881.601,E2 -27881.601} C_VEL
LIN {X 0,Y 154.479,Z 398.891,A -85,B 0,C 180,E1 -27882.395,E2 -27882.395} C_VEL
LIN {X 0,Y 152.779,Z 394.066,A -85,B 0,C 180,E1 -27885.345,E2 -27885.345} C_VEL
LIN {X 0,Y 151.117,Z 389.69,A -85,B 0,C 180,E1 -27888.941,E2 -27888.941} C_VEL
LIN {X 0,Y 149.629,Z 385.977,A -85,B 0,C 180,E1 -27893.596,E2 -27893.596} C_VEL
LIN {X 0,Y 148.976,Z 384.591,A -85,B 0,C 180,E1 -27897.297,E2 -27897.297} C_VEL
LIN {X 0,Y 148.856,Z 383.888,A -85,B 0,C 180,E1 -27900.001,E2 -27900.001} C_VEL
LIN {X 0,Y 149.108,Z 385.424,A -85,B 0,C 180,E1 -27904.648,E2 -27904.648} C_VEL
LIN {X 0,Y 149.956,Z 387.904,A -85,B 0,C 180,E1 -27908.592,E2 -27908.592} C_VEL
LIN {X 0,Y 151.425,Z 392.148,A -85,B 0,C 180,E1 -27912.737,E2 -27912.737} C_VEL
LIN {X 0,Y 153.013,Z 396.797,A -85,B 0,C 180,E1 -27915.998,E2 -27915.998} C_VEL
LIN {X 0,Y 154.783,Z 402.841,A -85,B 0,C 180,E1 -27919.048,E2 -27919.048} C_VEL
LIN {X 0,Y 155.07,Z 403.902,A -85,B 0,C 180,E1 -27919.503,E2 -27919.503} C_VEL
LIN {X 0,Y 152.266,Z 429.098,A -85,B 0,C 180,E1 -27920.2,E2 -27920.2} C_VEL
LIN {X 0,Y 149.43,Z 443.02,A -85,B 0,C 180,E1 -27920.816,E2 -27920.816} C_VEL
LIN {X 0,Y 145.927,Z 454.781,A -85,B 0,C 180,E1 -27921.551,E2 -27921.551} C_VEL
LIN {X 0,Y 140.947,Z 467.551,A -85,B 0,C 180,E1 -27922.713,E2 -27922.713} C_VEL
LIN {X 0,Y 134.906,Z 479.737,A -85,B 0,C 180,E1 -27924.264,E2 -27924.264} C_VEL
LIN {X 0,Y 128.553,Z 490.213,A -85,B 0,C 180,E1 -27926.105,E2 -27926.105} C_VEL
LIN {X 0,Y 121.72,Z 499.676,A -85,B 0,C 180,E1 -27928.296,E2 -27928.296} C_VEL
LIN {X 0,Y 113.196,Z 509.546,A -85,B 0,C 180,E1 -27931.385,E2 -27931.385} C_VEL
LIN {X 0,Y 105.133,Z 517.59,A -85,B 0,C 180,E1 -27935.027,E2 -27935.027} C_VEL
LIN {X 0,Y 96.302,Z 525.153,A -85,B 0,C 180,E1 -27939.98,E2 -27939.98} C_VEL
LIN {X 0,Y 89.453,Z 530.278,A -85,B 0,C 180,E1 -27945.002,E2 -27945.002} C_VEL
LIN {X 0,Y 83.466,Z 534.336,A -85,B 0,C 180,E1 -27950.839,E2 -27950.839} C_VEL
LIN {X 0,Y 78.295,Z 537.443,A -85,B 0,C 180,E1 -27957.413,E2 -27957.413} C_VEL
LIN {X 0,Y 73.218,Z 540.22,A -85,B 0,C 180,E1 -27967.421,E2 -27967.421} C_VEL
LIN {X 0,Y 70.385,Z 541.515,A -85,B 0,C 180,E1 -27978.48,E2 -27978.48} C_VEL
LIN {X 0,Y 69.758,Z 541.342,A -85,B 0,C 180,E1 -27990,E2 -27990} C_VEL
LIN {X 0,Y 70.209,Z 540.728,A -85,B 0,C 180,E1 -27995.745,E2 -27995.745} C_VEL
LIN {X 0,Y 72.581,Z 538.434,A -85,B 0,C 180,E1 -28006.887,E2 -28006.887} C_VEL
LIN {X 0,Y 75.8,Z 535.696,A -85,B 0,C 180,E1 -28014.659,E2 -28014.659} C_VEL
LIN {X 0,Y 81.939,Z 530.638,A -85,B 0,C 180,E1 -28023.883,E2 -28023.883} C_VEL
LIN {X 0,Y 87.696,Z 525.605,A -85,B 0,C 180,E1 -28029.874,E2 -28029.874} C_VEL
LIN {X 0,Y 95.389,Z 518.24,A -85,B 0,C 180,E1 -28035.917,E2 -28035.917} C_VEL
LIN {X 0,Y 102.729,Z 510.373,A -85,B 0,C 180,E1 -28040.321,E2 -28040.321} C_VEL
LIN {X 0,Y 110.516,Z 500.722,A -85,B 0,C 180,E1 -28044.173,E2 -28044.173} C_VEL
LIN {X 0,Y 116.7,Z 491.946,A -85,B 0,C 180,E1 -28046.676,E2 -28046.676} C_VEL
LIN {X 0,Y 122.302,Z 482.673,A -85,B 0,C 180,E1 -28048.72,E2 -28048.72} C_VEL
LIN {X 0,Y 128.027,Z 471.475,A -85,B 0,C 180,E1 -28050.545,E2 -28050.545} C_VEL
LIN {X 0,Y 133.218,Z 458.775,A -85,B 0,C 180,E1 -28052.084,E2 -28052.084} C_VEL
LIN {X 0,Y 137.246,Z 445.808,A -85,B 0,C 180,E1 -28053.192,E2 -28053.192} C_VEL
LIN {X 0,Y 140.043,Z 433.117,A -85,B 0,C 180,E1 -28053.901,E2 -28053.901} C_VEL
LIN {X 0,Y 142.165,Z 416.656,A -85,B 0,C 180,E1 -28054.447,E2 -28054.447} C_VEL
LIN {X 0,Y 144.367,Z 394.283,A -85,B 0,C 180,E1 -28055.154,E2 -28055.154} C_VEL
LIN {X 0,Y 142.052,Z 386.786,A -85,B 0,C 180,E1 -28058.596,E2 -28058.596} C_VEL
LIN {X 0,Y 140.155,Z 381.341,A -85,B 0,C 180,E1 -28061.923,E2 -28061.923} C_VEL
LIN {X 0,Y 138.502,Z 377.158,A -85,B 0,C 180,E1 -28065.525,E2 -28065.525} C_VEL
LIN {X 0,Y 137.167,Z 373.597,A -85,B 0,C 180,E1 -28069.668,E2 -28069.668} C_VEL
LIN {X 0,Y 136.191,Z 370.874,A -85,B 0,C 180,E1 -28076.323,E2 -28076.323} C_VEL
LIN {X 0,Y 136.304,Z 370.729,A -85,B 0,C 180,E1 -28080.368,E2 -28080.368} C_VEL
LIN {X 0,Y 137.393,Z 373.095,A -85,B 0,C 180,E1 -28086.285,E2 -28086.285} C_VEL
LIN {X 0,Y 139.258,Z 377.389,A -85,B 0,C 180,E1 -28091.369,E2 -28091.369} C_VEL
LIN {X 0,Y 140.927,Z 381.427,A -85,B 0,C 180,E1 -28094.646,E2 -28094.646} C_VEL
LIN {X 0,Y 143.251,Z 387.613,A -85,B 0,C 180,E1 -28098.364,E2 -28098.364} C_VEL
LIN {X 0,Y 144.701,Z 391.988,A -85,B 0,C 180,E1 -28100.403,E2 -28100.403} C_VEL
LIN {X 0,Y 140.56,Z 430.166,A -85,B 0,C 180,E1 -28101.585,E2 -28101.585} C_VEL
LIN {X 0,Y 137.719,Z 444.23,A -85,B 0,C 180,E1 -28102.296,E2 -28102.296} C_VEL
LIN {X 0,Y 133.84,Z 457.241,A -85,B 0,C 180,E1 -28103.232,E2 -28103.232} C_VEL
LIN {X 0,Y 128.622,Z 470.701,A -85,B 0,C 180,E1 -28104.718,E2 -28104.718} C_VEL
LIN {X 0,Y 122.694,Z 482.593,A -85,B 0,C 180,E1 -28106.493,E2 -28106.493} C_VEL
LIN {X 0,Y 116.615,Z 492.958,A -85,B 0,C 180,E1 -28108.683,E2 -28108.683} C_VEL
LIN {X 0,Y 109.359,Z 503.374,A -85,B 0,C 180,E1 -28111.625,E2 -28111.625} C_VEL
LIN {X 0,Y 101.375,Z 513.154,A -85,B 0,C 180,E1 -28115.455,E2 -28115.455} C_VEL
LIN {X 0,Y 93.981,Z 521.161,A -85,B 0,C 180,E1 -28119.961,E2 -28119.961} C_VEL
LIN {X 0,Y 86.258,Z 528.706,A -85,B 0,C 180,E1 -28126.169,E2 -28126.169} C_VEL
LIN {X 0,Y 80.676,Z 533.894,A -85,B 0,C 180,E1 -28132.427,E2 -28132.427} C_VEL
LIN {X 0,Y 76.037,Z 538,A -85,B 0,C 180,E1 -28139.446,E2 -28139.446} C_VEL
LIN {X 0,Y 72.505,Z 541.156,A -85,B 0,C 180,E1 -28147.188,E2 -28147.188} C_VEL
LIN {X 0,Y 69.992,Z 544.024,A -85,B 0,C 180,E1 -28158.416,E2 -28158.416} C_VEL
LIN {X 0,Y 69.564,Z 544.901,A -85,B 0,C 180,E1 -28164.202,E2 -28164.202} C_VEL
LIN {X 0,Y 69.667,Z 545.397,A -85,B 0,C 180,E1 -28170,E2 -28170} C_VEL
LIN {X 0,Y 69.585,Z 545.496,A -85,B 0,C 180,E1 -28175.797,E2 -28175.797} C_VEL
LIN {X 0,Y 71.021,Z 544.614,A -85,B 0,C 180,E1 -28187.27,E2 -28187.27} C_VEL
LIN {X 0,Y 74.825,Z 542.289,A -85,B 0,C 180,E1 -28198.01,E2 -28198.01} C_VEL
LIN {X 0,Y 80.888,Z 538.465,A -85,B 0,C 180,E1 -28207.459,E2 -28207.459} C_VEL
LIN {X 0,Y 86.544,Z 534.472,A -85,B 0,C 180,E1 -28213.65,E2 -28213.65} C_VEL
LIN {X 0,Y 93.141,Z 529.477,A -85,B 0,C 180,E1 -28218.985,E2 -28218.985} C_VEL
LIN {X 0,Y 101.73,Z 522.22,A -85,B 0,C 180,E1 -28224.266,E2 -28224.266} C_VEL
LIN {X 0,Y 109.768,Z 514.518,A -85,B 0,C 180,E1 -28228.031,E2 -28228.031} C_VEL
LIN {X 0,Y 118.139,Z 505.101,A -85,B 0,C 180,E1 -28231.336,E2 -28231.336} C_VEL
LIN {X 0,Y 126.066,Z 494.507,A -85,B 0,C 180,E1 -28234.018,E2 -28234.018} C_VEL
LIN {X 0,Y 133.567,Z 482.653,A -85,B 0,C 180,E1 -28236.095,E2 -28236.095} C_VEL
LIN {X 0,Y 139.645,Z 470.843,A -85,B 0,C 180,E1 -28237.632,E2 -28237.632} C_VEL
LIN {X 0,Y 145.093,Z 457.524,A -85,B 0,C 180,E1 -28238.814,E2 -28238.814} C_VEL
LIN {X 0,Y 149.401,Z 443.31,A -85,B 0,C 180,E1 -28239.697,E2 -28239.697} C_VEL
LIN {X 0,Y 152.222,Z 429.448,A -85,B 0,C 180,E1 -28240.279,E2 -28240.279} C_VEL
LIN {X 0,Y 155.346,Z 401.599,A -85,B 0,C 180,E1 -28241.047,E2 -28241.047} C_VEL
LIN {X 0,Y 154.479,Z 398.891,A -85,B 0,C 180,E1 -28242.395,E2 -28242.395} C_VEL
LIN {X 0,Y 153.693,Z 396.979,A -85,B 0,C 180,E1 -28243.637,E2 -28243.637} C_VEL
LIN {X 0,Y 152.391,Z 395.196,A -85,B 0,C 180,E1 -28245.694,E2 -28245.694} C_VEL
LIN {X 0,Y 150.333,Z 394.039,A -85,B 0,C 180,E1 -28249.395,E2 -28249.395} C_VEL
LIN {X 0,Y 148.642,Z 392.915,A -85,B 0,C 180,E1 -28254.033,E2 -28254.033} C_VEL
LIN {X 0,Y 148.109,Z 391.659,A -85,B 0,C 180,E1 -28257.281,E2 -28257.281} C_VEL
LIN {X 0,Y 147.987,Z 390.962,A -85,B 0,C 180,E1 -28260.001,E2 -28260.001} C_VEL
LIN {X 0,Y 148.175,Z 392.389,A -85,B 0,C 180,E1 -28264.251,E2 -28264.251} C_VEL
LIN {X 0,Y 148.847,Z 394.667,A -85,B 0,C 180,E1 -28267.855,E2 -28267.855} C_VEL
LIN {X 0,Y 150.094,Z 398.728,A -85,B 0,C 180,E1 -28271.822,E2 -28271.822} C_VEL
LIN {X 0,Y 151.38,Z 402.934,A -85,B 0,C 180,E1 -28274.795,E2 -28274.795} C_VEL
LIN {X 0,Y 152.514,Z 407.263,A -85,B 0,C 180,E1 -28277.06,E2 -28277.06} C_VEL
LIN {X 0,Y 149.858,Z 429.92,A -85,B 0,C 180,E1 -28277.688,E2 -28277.688} C_VEL
LIN {X 0,Y 146.733,Z 444.341,A -85,B 0,C 180,E1 -28278.276,E2 -28278.276} C_VEL
LIN {X 0,Y 142.602,Z 457.337,A -85,B 0,C 180,E1 -28279.073,E2 -28279.073} C_VEL
LIN {X 0,Y 137.585,Z 469.381,A -85,B 0,C 180,E1 -28280.182,E2 -28280.182} C_VEL
LIN {X 0,Y 131.372,Z 481.137,A -85,B 0,C 180,E1 -28281.644,E2 -28281.644} C_VEL
LIN {X 0,Y 124.166,Z 492.355,A -85,B 0,C 180,E1 -28283.621,E2 -28283.621} C_VEL
LIN {X 0,Y 115.531,Z 503.34,A -85,B 0,C 180,E1 -28286.199,E2 -28286.199} C_VEL
LIN {X 0,Y 106.8,Z 512.55,A -85,B 0,C 180,E1 -28289.319,E2 -28289.319} C_VEL
LIN {X 0,Y 98.482,Z 520.067,A -85,B 0,C 180,E1 -28293.017,E2 -28293.017} C_VEL
LIN {X 0,Y 89.376,Z 527.105,A -85,B 0,C 180,E1 -28298.156,E2 -28298.156} C_VEL
LIN {X 0,Y 82.991,Z 531.456,A -85,B 0,C 180,E1 -28302.896,E2 -28302.896} C_VEL
LIN {X 0,Y 76.114,Z 535.641,A -85,B 0,C 180,E1 -28309.734,E2 -28309.734} C_VEL
LIN {X 0,Y 69.22,Z 539.195,A -85,B 0,C 180,E1 -28319.492,E2 -28319.492} C_VEL
LIN {X 0,Y 64.764,Z 541.242,A -85,B 0,C 180,E1 -28331.001,E2 -28331.001} C_VEL
LIN {X 0,Y 62.756,Z 541.806,A -85,B 0,C 180,E1 -28343.57,E2 -28343.57} C_VEL
LIN {X 0,Y 62.68,Z 541.548,A -85,B 0,C 180,E1 -28350,E2 -28350} C_VEL
LIN {X 0,Y 63.152,Z 540.941,A -85,B 0,C 180,E1 -28356.389,E2 -28356.389} C_VEL
LIN {X 0,Y 65.837,Z 538.658,A -85,B 0,C 180,E1 -28368.677,E2 -28368.677} C_VEL
LIN {X 0,Y 69.431,Z 535.933,A -85,B 0,C 180,E1 -28377.096,E2 -28377.096} C_VEL
LIN {X 0,Y 76.147,Z 530.893,A -85,B 0,C 180,E1 -28386.863,E2 -28386.863} C_VEL
LIN {X 0,Y 82.393,Z 525.874,A -85,B 0,C 180,E1 -28393.029,E2 -28393.029} C_VEL
LIN {X 0,Y 90.597,Z 518.543,A -85,B 0,C 180,E1 -28399.142,E2 -28399.142} C_VEL
LIN {X 0,Y 98.364,Z 510.701,A -85,B 0,C 180,E1 -28403.493,E2 -28403.493} C_VEL
LIN {X 0,Y 106.528,Z 501.084,A -85,B 0,C 180,E1 -28407.261,E2 -28407.261} C_VEL
LIN {X 0,Y 112.961,Z 492.353,A -85,B 0,C 180,E1 -28409.681,E2 -28409.681} C_VEL
LIN {X 0,Y 118.732,Z 483.217,A -85,B 0,C 180,E1 -28411.627,E2 -28411.627} C_VEL
LIN {X 0,Y 124.697,Z 472.017,A -85,B 0,C 180,E1 -28413.38,E2 -28413.38} C_VEL
LIN {X 0,Y 130.063,Z 459.429,A -85,B 0,C 180,E1 -28414.833,E2 -28414.833} C_VEL
LIN {X 0,Y 134.462,Z 445.757,A -85,B 0,C 180,E1 -28415.95,E2 -28415.95} C_VEL
LIN {X 0,Y 137.5,Z 432.111,A -85,B 0,C 180,E1 -28416.641,E2 -28416.641} C_VEL
LIN {X 0,Y 139.854,Z 413.24,A -85,B 0,C 180,E1 -28417.229,E2 -28417.229} C_VEL
LIN {X 0,Y 141.448,Z 397.373,A -85,B 0,C 180,E1 -28417.735,E2 -28417.735} C_VEL
LIN {X 0,Y 139.349,Z 390.02,A -85,B 0,C 180,E1 -28421.509,E2 -28421.509} C_VEL
LIN {X 0,Y 137.826,Z 385.577,A -85,B 0,C 180,E1 -28424.812,E2 -28424.812} C_VEL
LIN {X 0,Y 137.075,Z 383.427,A -85,B 0,C 180,E1 -28426.831,E2 -28426.831} C_VEL
LIN {X 0,Y 136.014,Z 380.261,A -85,B 0,C 180,E1 -28430.707,E2 -28430.707} C_VEL
LIN {X 0,Y 135.314,Z 377.873,A -85,B 0,C 180,E1 -28436.66,E2 -28436.66} C_VEL
LIN {X 0,Y 135.43,Z 377.845,A -85,B 0,C 180,E1 -28440.371,E2 -28440.371} C_VEL
LIN {X 0,Y 136.311,Z 379.979,A -85,B 0,C 180,E1 -28445.653,E2 -28445.653} C_VEL
LIN {X 0,Y 137.893,Z 384.057,A -85,B 0,C 180,E1 -28450.46,E2 -28450.46} C_VEL
LIN {X 0,Y 139.421,Z 388.113,A -85,B 0,C 180,E1 -28453.76,E2 -28453.76} C_VEL
LIN {X 0,Y 141.285,Z 393.75,A -85,B 0,C 180,E1 -28457.085,E2 -28457.085} C_VEL
LIN {X 0,Y 141.744,Z 395.225,A -85,B 0,C 180,E1 -28457.823,E2 -28457.823} C_VEL
LIN {X 0,Y 137.869,Z 430.091,A -85,B 0,C 180,E1 -28458.888,E2 -28458.888} C_VEL
LIN {X 0,Y 135.024,Z 443.87,A -85,B 0,C 180,E1 -28459.537,E2 -28459.537} C_VEL
LIN {X 0,Y 130.796,Z 457.643,A -85,B 0,C 180,E1 -28460.456,E2 -28460.456} C_VEL
LIN {X 0,Y 125.801,Z 470.131,A -85,B 0,C 180,E1 -28461.759,E2 -28461.759} C_VEL
LIN {X 0,Y 119.687,Z 482.132,A -85,B 0,C 180,E1 -28463.44,E2 -28463.44} C_VEL
LIN {X 0,Y 112.781,Z 493.399,A -85,B 0,C 180,E1 -28465.711,E2 -28465.711} C_VEL
LIN {X 0,Y 105.792,Z 503.012,A -85,B 0,C 180,E1 -28468.332,E2 -28468.332} C_VEL
LIN {X 0,Y 97.412,Z 512.826,A -85,B 0,C 180,E1 -28472.037,E2 -28472.037} C_VEL
LIN {X 0,Y 89.56,Z 520.859,A -85,B 0,C 180,E1 -28476.455,E2 -28476.455} C_VEL
LIN {X 0,Y 81.241,Z 528.435,A -85,B 0,C 180,E1 -28482.668,E2 -28482.668} C_VEL
LIN {X 0,Y 75.112,Z 533.633,A -85,B 0,C 180,E1 -28489.084,E2 -28489.084} C_VEL
LIN {X 0,Y 69.971,Z 537.753,A -85,B 0,C 180,E1 -28496.467,E2 -28496.467} C_VEL
LIN {X 0,Y 65.975,Z 540.923,A -85,B 0,C 180,E1 -28504.78,E2 -28504.78} C_VEL
LIN {X 0,Y 63.009,Z 543.804,A -85,B 0,C 180,E1 -28517.111,E2 -28517.111} C_VEL
LIN {X 0,Y 62.502,Z 544.688,A -85,B 0,C 180,E1 -28523.544,E2 -28523.544} C_VEL
LIN {X 0,Y 62.557,Z 545.194,A -85,B 0,C 180,E1 -28530,E2 -28530} C_VEL
LIN {X 0,Y 62.519,Z 545.3,A -85,B 0,C 180,E1 -28536.455,E2 -28536.455} C_VEL
LIN {X 0,Y 64.221,Z 544.426,A -85,B 0,C 180,E1 -28549.166,E2 -28549.166} C_VEL
LIN {X 0,Y 68.589,Z 542.113,A -85,B 0,C 180,E1 -28560.819,E2 -28560.819} C_VEL
LIN {X 0,Y 75.322,Z 538.3,A -85,B 0,C 180,E1 -28570.779,E2 -28570.779} C_VEL
LIN {X 0,Y 81.519,Z 534.316,A -85,B 0,C 180,E1 -28577.122,E2 -28577.122} C_VEL
LIN {X 0,Y 88.612,Z 529.33,A -85,B 0,C 180,E1 -28582.477,E2 -28582.477} C_VEL
LIN {X 0,Y 97.735,Z 522.083,A -85,B 0,C 180,E1 -28587.663,E2 -28587.663} C_VEL
LIN {X 0,Y 106.175,Z 514.39,A -85,B 0,C 180,E1 -28591.287,E2 -28591.287} C_VEL
LIN {X 0,Y 114.191,Z 505.814,A -85,B 0,C 180,E1 -28594.221,E2 -28594.221} C_VEL
LIN {X 0,Y 122.353,Z 495.469,A -85,B 0,C 180,E1 -28596.785,E2 -28596.785} C_VEL
LIN {X 0,Y 130.074,Z 483.84,A -85,B 0,C 180,E1 -28598.751,E2 -28598.751} C_VEL
LIN {X 0,Y 136.316,Z 472.324,A -85,B 0,C 180,E1 -28600.202,E2 -28600.202} C_VEL
LIN {X 0,Y 141.892,Z 459.593,A -85,B 0,C 180,E1 -28601.309,E2 -28601.309} C_VEL
LIN {X 0,Y 146.279,Z 446.224,A -85,B 0,C 180,E1 -28602.153,E2 -28602.153} C_VEL
LIN {X 0,Y 149.449,Z 432.28,A -85,B 0,C 180,E1 -28602.733,E2 -28602.733} C_VEL
LIN {X 0,Y 152.004,Z 412.464,A -85,B 0,C 180,E1 -28603.24,E2 -28603.24} C_VEL
LIN {X 0,Y 152.757,Z 405.146,A -85,B 0,C 180,E1 -28603.484,E2 -28603.484} C_VEL
LIN {X 0,Y 151.028,Z 399.697,A -85,B 0,C 180,E1 -28606.889,E2 -28606.889} C_VEL
LIN {X 0,Y 149.588,Z 395.648,A -85,B 0,C 180,E1 -28610.538,E2 -28610.538} C_VEL
LIN {X 0,Y 148.642,Z 392.915,A -85,B 0,C 180,E1 -28614.033,E2 -28614.033} C_VEL
LIN {X 0,Y 148.299,Z 392.622,A -85,B 0,C 180,E1 -28615.541,E2 -28615.541} C_VEL
LIN {X 0,Y 147.829,Z 393.414,A -85,B 0,C 180,E1 -28617.809,E2 -28617.809} C_VEL
LIN {X 0,Y 147.331,Z 396.623,A -85,B 0,C 180,E1 -28621.515,E2 -28621.515} C_VEL
LIN {X 0,Y 147.346,Z 399.51,A -85,B 0,C 180,E1 -28624.502,E2 -28624.502} C_VEL
LIN {X 0,Y 147.555,Z 400.623,A -85,B 0,C 180,E1 -28626.031,E2 -28626.031} C_VEL
LIN {X 0,Y 148.611,Z 404.525,A -85,B 0,C 180,E1 -28630.302,E2 -28630.302} C_VEL
LIN {X 0,Y 149.803,Z 409.08,A -85,B 0,C 180,E1 -28633.568,E2 -28633.568} C_VEL
LIN {X 0,Y 150.214,Z 410.83,A -85,B 0,C 180,E1 -28634.548,E2 -28634.548} C_VEL
LIN {X 0,Y 147.885,Z 429.903,A -85,B 0,C 180,E1 -28635.059,E2 -28635.059} C_VEL
LIN {X 0,Y 144.846,Z 443.841,A -85,B 0,C 180,E1 -28635.601,E2 -28635.601} C_VEL
LIN {X 0,Y 140.735,Z 456.65,A -85,B 0,C 180,E1 -28636.296,E2 -28636.296} C_VEL
LIN {X 0,Y 135.303,Z 469.482,A -85,B 0,C 180,E1 -28637.364,E2 -28637.364} C_VEL
LIN {X 0,Y 128.923,Z 481.24,A -85,B 0,C 180,E1 -28638.711,E2 -28638.711} C_VEL
LIN {X 0,Y 121.281,Z 492.754,A -85,B 0,C 180,E1 -28640.606,E2 -28640.606} C_VEL
LIN {X 0,Y 112.577,Z 503.455,A -85,B 0,C 180,E1 -28642.956,E2 -28642.956} C_VEL
LIN {X 0,Y 103.498,Z 512.676,A -85,B 0,C 180,E1 -28645.878,E2 -28645.878} C_VEL
LIN {X 0,Y 94.795,Z 520.202,A -85,B 0,C 180,E1 -28649.411,E2 -28649.411} C_VEL
LIN {X 0,Y 85.152,Z 527.249,A -85,B 0,C 180,E1 -28654.377,E2 -28654.377} C_VEL
LIN {X 0,Y 77.753,Z 531.934,A -85,B 0,C 180,E1 -28659.504,E2 -28659.504} C_VEL
LIN {X 0,Y 70.813,Z 535.806,A -85,B 0,C 180,E1 -28665.995,E2 -28665.995} C_VEL
LIN {X 0,Y 63.177,Z 539.371,A -85,B 0,C 180,E1 -28676.206,E2 -28676.206} C_VEL
LIN {X 0,Y 58.087,Z 541.428,A -85,B 0,C 180,E1 -28688.717,E2 -28688.717} C_VEL
LIN {X 0,Y 55.693,Z 542.008,A -85,B 0,C 180,E1 -28702.75,E2 -28702.75} C_VEL
LIN {X 0,Y 55.592,Z 541.755,A -85,B 0,C 180,E1 -28710,E2 -28710} C_VEL
LIN {X 0,Y 56.118,Z 541.154,A -85,B 0,C 180,E1 -28717.194,E2 -28717.194} C_VEL
LIN {X 0,Y 59.165,Z 538.883,A -85,B 0,C 180,E1 -28730.876,E2 -28730.876} C_VEL
LIN {X 0,Y 63.195,Z 536.171,A -85,B 0,C 180,E1 -28740.029,E2 -28740.029} C_VEL
LIN {X 0,Y 70.595,Z 531.146,A -85,B 0,C 180,E1 -28750.322,E2 -28750.322} C_VEL
LIN {X 0,Y 77.362,Z 526.144,A -85,B 0,C 180,E1 -28756.615,E2 -28756.615} C_VEL
LIN {X 0,Y 86.129,Z 518.844,A -85,B 0,C 180,E1 -28762.709,E2 -28762.709} C_VEL
LIN {X 0,Y 94.326,Z 511.029,A -85,B 0,C 180,E1 -28766.95,E2 -28766.95} C_VEL
LIN {X 0,Y 102.874,Z 501.446,A -85,B 0,C 180,E1 -28770.577,E2 -28770.577} C_VEL
LIN {X 0,Y 109.555,Z 492.758,A -85,B 0,C 180,E1 -28772.881,E2 -28772.881} C_VEL
LIN {X 0,Y 116.388,Z 482.287,A -85,B 0,C 180,E1 -28774.924,E2 -28774.924} C_VEL
LIN {X 0,Y 122.547,Z 470.825,A -85,B 0,C 180,E1 -28776.574,E2 -28776.574} C_VEL
LIN {X 0,Y 128.002,Z 458.096,A -85,B 0,C 180,E1 -28777.897,E2 -28777.897} C_VEL
LIN {X 0,Y 132.137,Z 445.185,A -85,B 0,C 180,E1 -28778.848,E2 -28778.848} C_VEL
LIN {X 0,Y 135.287,Z 430.992,A -85,B 0,C 180,E1 -28779.502,E2 -28779.502} C_VEL
LIN {X 0,Y 138.056,Z 408.227,A -85,B 0,C 180,E1 -28780.134,E2 -28780.134} C_VEL
LIN {X 0,Y 138.827,Z 400.714,A -85,B 0,C 180,E1 -28780.376,E2 -28780.376} C_VEL
LIN {X 0,Y 137.402,Z 395.233,A -85,B 0,C 180,E1 -28783.462,E2 -28783.462} C_VEL
LIN {X 0,Y 136.031,Z 390.58,A -85,B 0,C 180,E1 -28787.165,E2 -28787.165} C_VEL
LIN {X 0,Y 134.975,Z 387.058,A -85,B 0,C 180,E1 -28791.429,E2 -28791.429} C_VEL
LIN {X 0,Y 134.443,Z 384.873,A -85,B 0,C 180,E1 -28797.002,E2 -28797.002} C_VEL
LIN {X 0,Y 134.555,Z 384.964,A -85,B 0,C 180,E1 -28800.373,E2 -28800.373} C_VEL
LIN {X 0,Y 135.232,Z 386.77,A -85,B 0,C 180,E1 -28804.899,E2 -28804.899} C_VEL
LIN {X 0,Y 136.56,Z 390.663,A -85,B 0,C 180,E1 -28809.511,E2 -28809.511} C_VEL
LIN {X 0,Y 137.836,Z 394.439,A -85,B 0,C 180,E1 -28812.608,E2 -28812.608} C_VEL
LIN {X 0,Y 139.082,Z 398.667,A -85,B 0,C 180,E1 -28815.168,E2 -28815.168} C_VEL
LIN {X 0,Y 135.578,Z 429.574,A -85,B 0,C 180,E1 -28816.08,E2 -28816.08} C_VEL
LIN {X 0,Y 132.636,Z 443.533,A -85,B 0,C 180,E1 -28816.66,E2 -28816.66} C_VEL
LIN {X 0,Y 128.486,Z 456.913,A -85,B 0,C 180,E1 -28817.487,E2 -28817.487} C_VEL
LIN {X 0,Y 123.339,Z 469.542,A -85,B 0,C 180,E1 -28818.685,E2 -28818.685} C_VEL
LIN {X 0,Y 117.042,Z 481.671,A -85,B 0,C 180,E1 -28820.246,E2 -28820.246} C_VEL
LIN {X 0,Y 110.651,Z 491.884,A -85,B 0,C 180,E1 -28822.104,E2 -28822.104} C_VEL
LIN {X 0,Y 102.603,Z 502.65,A -85,B 0,C 180,E1 -28824.829,E2 -28824.829} C_VEL
LIN {X 0,Y 93.819,Z 512.497,A -85,B 0,C 180,E1 -28828.337,E2 -28828.337} C_VEL
LIN {X 0,Y 85.507,Z 520.556,A -85,B 0,C 180,E1 -28832.601,E2 -28832.601} C_VEL
LIN {X 0,Y 76.567,Z 528.163,A -85,B 0,C 180,E1 -28838.722,E2 -28838.722} C_VEL
LIN {X 0,Y 69.834,Z 533.371,A -85,B 0,C 180,E1 -28845.215,E2 -28845.215} C_VEL
LIN {X 0,Y 64.131,Z 537.507,A -85,B 0,C 180,E1 -28852.935,E2 -28852.935} C_VEL
LIN {X 0,Y 59.585,Z 540.69,A -85,B 0,C 180,E1 -28861.85,E2 -28861.85} C_VEL
LIN {X 0,Y 56.074,Z 543.584,A -85,B 0,C 180,E1 -28875.484,E2 -28875.484} C_VEL
LIN {X 0,Y 55.437,Z 544.475,A -85,B 0,C 180,E1 -28882.717,E2 -28882.717} C_VEL
LIN {X 0,Y 55.468,Z 544.991,A -85,B 0,C 180,E1 -28890,E2 -28890} C_VEL
LIN {X 0,Y 55.454,Z 545.103,A -85,B 0,C 180,E1 -28897.281,E2 -28897.281} C_VEL
LIN {X 0,Y 57.519,Z 544.24,A -85,B 0,C 180,E1 -28911.503,E2 -28911.503} C_VEL
LIN {X 0,Y 62.554,Z 541.937,A -85,B 0,C 180,E1 -28924.177,E2 -28924.177} C_VEL
LIN {X 0,Y 70.042,Z 538.134,A -85,B 0,C 180,E1 -28934.617,E2 -28934.617} C_VEL
LIN {X 0,Y 76.826,Z 534.159,A -85,B 0,C 180,E1 -28941.038,E2 -28941.038} C_VEL
LIN {X 0,Y 84.454,Z 529.184,A -85,B 0,C 180,E1 -28946.322,E2 -28946.322} C_VEL
LIN {X 0,Y 94.116,Z 521.946,A -85,B 0,C 180,E1 -28951.33,E2 -28951.33} C_VEL
LIN {X 0,Y 102.948,Z 514.262,A -85,B 0,C 180,E1 -28954.76,E2 -28954.76} C_VEL
LIN {X 0,Y 111.738,Z 505.172,A -85,B 0,C 180,E1 -28957.672,E2 -28957.672} C_VEL
LIN {X 0,Y 120.512,Z 494.285,A -85,B 0,C 180,E1 -28960.112,E2 -28960.112} C_VEL
LIN {X 0,Y 128.462,Z 482.439,A -85,B 0,C 180,E1 -28961.907,E2 -28961.907} C_VEL
LIN {X 0,Y 134.888,Z 470.633,A -85,B 0,C 180,E1 -28963.209,E2 -28963.209} C_VEL
LIN {X 0,Y 140.509,Z 457.507,A -85,B 0,C 180,E1 -28964.211,E2 -28964.211} C_VEL
LIN {X 0,Y 144.947,Z 443.58,A -85,B 0,C 180,E1 -28964.939,E2 -28964.939} C_VEL
LIN {X 0,Y 147.955,Z 429.591,A -85,B 0,C 180,E1 -28965.437,E2 -28965.437} C_VEL
LIN {X 0,Y 150.452,Z 409.104,A -85,B 0,C 180,E1 -28965.922,E2 -28965.922} C_VEL
LIN {X 0,Y 149.125,Z 404.639,A -85,B 0,C 180,E1 -28969.135,E2 -28969.135} C_VEL
LIN {X 0,Y 148.26,Z 401.967,A -85,B 0,C 180,E1 -28971.825,E2 -28971.825} C_VEL
LIN {X 0,Y 147.584,Z 399.663,A -85,B 0,C 180,E1 -28974.878,E2 -28974.878} C_VEL
LIN {X 0,Y 147.178,Z 398.566,A -85,B 0,C 180,E1 -28977.948,E2 -28977.948} C_VEL
LIN {X 0,Y 147.117,Z 398.047,A -85,B 0,C 180,E1 -28980.001,E2 -28980.001} C_VEL
LIN {X 0,Y 147.24,Z 399.316,A -85,B 0,C 180,E1 -28983.764,E2 -28983.764} C_VEL
LIN {X 0,Y 147.555,Z 400.623,A -85,B 0,C 180,E1 -28986.031,E2 -28986.031} C_VEL
LIN {X 0,Y 147.94,Z 402.644,A -85,B 0,C 180,E1 -28988.086,E2 -28988.086} C_VEL
LIN {X 0,Y 148.253,Z 405.908,A -85,B 0,C 180,E1 -28989.889,E2 -28989.889} C_VEL
LIN {X 0,Y 148.374,Z 408.987,A -85,B 0,C 180,E1 -28990.974,E2 -28990.974} C_VEL
LIN {X 0,Y 148.321,Z 412.596,A -85,B 0,C 180,E1 -28991.755,E2 -28991.755} C_VEL
LIN {X 0,Y 148.138,Z 415.237,A -85,B 0,C 180,E1 -28992.033,E2 -28992.033} C_VEL
LIN {X 0,Y 145.805,Z 432.265,A -85,B 0,C 180,E1 -28992.436,E2 -28992.436} C_VEL
LIN {X 0,Y 142.879,Z 444.743,A -85,B 0,C 180,E1 -28992.879,E2 -28992.879} C_VEL
LIN {X 0,Y 138.806,Z 457.045,A -85,B 0,C 180,E1 -28993.504,E2 -28993.504} C_VEL
LIN {X 0,Y 133.361,Z 469.583,A -85,B 0,C 180,E1 -28994.458,E2 -28994.458} C_VEL
LIN {X 0,Y 126.824,Z 481.343,A -85,B 0,C 180,E1 -28995.672,E2 -28995.672} C_VEL
LIN {X 0,Y 118.761,Z 493.137,A -85,B 0,C 180,E1 -28997.449,E2 -28997.449} C_VEL
LIN {X 0,Y 110.005,Z 503.571,A -85,B 0,C 180,E1 -28999.552,E2 -28999.552} C_VEL
LIN {X 0,Y 100.598,Z 512.802,A -85,B 0,C 180,E1 -29002.232,E2 -29002.232} C_VEL
LIN {X 0,Y 91.512,Z 520.336,A -85,B 0,C 180,E1 -29005.529,E2 -29005.529} C_VEL
LIN {X 0,Y 81.346,Z 527.393,A -85,B 0,C 180,E1 -29010.236,E2 -29010.236} C_VEL
LIN {X 0,Y 74.182,Z 531.672,A -85,B 0,C 180,E1 -29014.644,E2 -29014.644} C_VEL
LIN {X 0,Y 65.855,Z 535.971,A -85,B 0,C 180,E1 -29021.666,E2 -29021.666} C_VEL
LIN {X 0,Y 57.388,Z 539.546,A -85,B 0,C 180,E1 -29032.243,E2 -29032.243} C_VEL
LIN {X 0,Y 51.505,Z 541.614,A -85,B 0,C 180,E1 -29045.836,E2 -29045.836} C_VEL
LIN {X 0,Y 49.671,Z 542.1,A -85,B 0,C 180,E1 -29053.562,E2 -29053.562} C_VEL
LIN {X 0,Y 48.493,Z 541.963,A -85,B 0,C 180,E1 -29070,E2 -29070} C_VEL
LIN {X 0,Y 49.091,Z 541.367,A -85,B 0,C 180,E1 -29078.23,E2 -29078.23} C_VEL
LIN {X 0,Y 52.59,Z 539.108,A -85,B 0,C 180,E1 -29093.634,E2 -29093.634} C_VEL
LIN {X 0,Y 59.01,Z 535.339,A -85,B 0,C 180,E1 -29106.546,E2 -29106.546} C_VEL
LIN {X 0,Y 65.349,Z 531.399,A -85,B 0,C 180,E1 -29114.349,E2 -29114.349} C_VEL
LIN {X 0,Y 72.677,Z 526.414,A -85,B 0,C 180,E1 -29120.678,E2 -29120.678} C_VEL
LIN {X 0,Y 82.034,Z 519.144,A -85,B 0,C 180,E1 -29126.646,E2 -29126.646} C_VEL
LIN {X 0,Y 90.661,Z 511.357,A -85,B 0,C 180,E1 -29130.7,E2 -29130.7} C_VEL
LIN {X 0,Y 99.59,Z 501.807,A -85,B 0,C 180,E1 -29134.124,E2 -29134.124} C_VEL
LIN {X 0,Y 106.519,Z 493.162,A -85,B 0,C 180,E1 -29136.268,E2 -29136.268} C_VEL
LIN {X 0,Y 113.573,Z 482.748,A -85,B 0,C 180,E1 -29138.155,E2 -29138.155} C_VEL
LIN {X 0,Y 119.911,Z 471.364,A -85,B 0,C 180,E1 -29139.676,E2 -29139.676} C_VEL
LIN {X 0,Y 125.513,Z 458.757,A -85,B 0,C 180,E1 -29140.888,E2 -29140.888} C_VEL
LIN {X 0,Y 129.959,Z 445.39,A -85,B 0,C 180,E1 -29141.794,E2 -29141.794} C_VEL
LIN {X 0,Y 133.005,Z 432.32,A -85,B 0,C 180,E1 -29142.342,E2 -29142.342} C_VEL
LIN {X 0,Y 135.389,Z 414.478,A -85,B 0,C 180,E1 -29142.818,E2 -29142.818} C_VEL
LIN {X 0,Y 136.484,Z 404.181,A -85,B 0,C 180,E1 -29143.133,E2 -29143.133} C_VEL
LIN {X 0,Y 135.467,Z 399.803,A -85,B 0,C 180,E1 -29145.924,E2 -29145.924} C_VEL
LIN {X 0,Y 134.618,Z 396.621,A -85,B 0,C 180,E1 -29148.794,E2 -29148.794} C_VEL
LIN {X 0,Y 133.967,Z 393.885,A -85,B 0,C 180,E1 -29152.107,E2 -29152.107} C_VEL
LIN {X 0,Y 133.573,Z 391.962,A -85,B 0,C 180,E1 -29156.983,E2 -29156.983} C_VEL
LIN {X 0,Y 133.681,Z 392.085,A -85,B 0,C 180,E1 -29160.376,E2 -29160.376} C_VEL
LIN {X 0,Y 134.199,Z 393.665,A -85,B 0,C 180,E1 -29164.251,E2 -29164.251} C_VEL
LIN {X 0,Y 135.231,Z 397.124,A -85,B 0,C 180,E1 -29168.404,E2 -29168.404} C_VEL
LIN {X 0,Y 136.231,Z 400.582,A -85,B 0,C 180,E1 -29171.248,E2 -29171.248} C_VEL
LIN {X 0,Y 136.704,Z 402.404,A -85,B 0,C 180,E1 -29172.43,E2 -29172.43} C_VEL
LIN {X 0,Y 133.433,Z 430.062,A -85,B 0,C 180,E1 -29173.202,E2 -29173.202} C_VEL
LIN {X 0,Y 130.418,Z 443.887,A -85,B 0,C 180,E1 -29173.732,E2 -29173.732} C_VEL
LIN {X 0,Y 126.115,Z 457.315,A -85,B 0,C 180,E1 -29174.481,E2 -29174.481} C_VEL
LIN {X 0,Y 120.428,Z 470.678,A -85,B 0,C 180,E1 -29175.657,E2 -29175.657} C_VEL
LIN {X 0,Y 113.956,Z 482.507,A -85,B 0,C 180,E1 -29177.077,E2 -29177.077} C_VEL
LIN {X 0,Y 106.525,Z 493.731,A -85,B 0,C 180,E1 -29179.063,E2 -29179.063} C_VEL
LIN {X 0,Y 98.263,Z 504.083,A -85,B 0,C 180,E1 -29181.601,E2 -29181.601} C_VEL
LIN {X 0,Y 89.154,Z 513.662,A -85,B 0,C 180,E1 -29184.971,E2 -29184.971} C_VEL
LIN {X 0,Y 80.464,Z 521.476,A -85,B 0,C 180,E1 -29189.142,E2 -29189.142} C_VEL
LIN {X 0,Y 72.313,Z 527.89,A -85,B 0,C 180,E1 -29194.301,E2 -29194.301} C_VEL
LIN {X 0,Y 64.925,Z 533.107,A -85,B 0,C 180,E1 -29200.737,E2 -29200.737} C_VEL
LIN {X 0,Y 58.574,Z 537.26,A -85,B 0,C 180,E1 -29208.708,E2 -29208.708} C_VEL
LIN {X 0,Y 53.387,Z 540.458,A -85,B 0,C 180,E1 -29218.227,E2 -29218.227} C_VEL
LIN {X 0,Y 49.208,Z 543.365,A -85,B 0,C 180,E1 -29233.403,E2 -29233.403} C_VEL
LIN {X 0,Y 48.381,Z 544.261,A -85,B 0,C 180,E1 -29241.648,E2 -29241.648} C_VEL
LIN {X 0,Y 48.362,Z 544.786,A -85,B 0,C 180,E1 -29250,E2 -29250} C_VEL
LIN {X 0,Y 48.397,Z 544.906,A -85,B 0,C 180,E1 -29258.35,E2 -29258.35} C_VEL
LIN {X 0,Y 50.946,Z 544.053,A -85,B 0,C 180,E1 -29274.447,E2 -29274.447} C_VEL
LIN {X 0,Y 56.784,Z 541.76,A -85,B 0,C 180,E1 -29288.231,E2 -29288.231} C_VEL
LIN {X 0,Y 65.118,Z 537.968,A -85,B 0,C 180,E1 -29299.067,E2 -29299.067} C_VEL
LIN {X 0,Y 72.535,Z 534.003,A -85,B 0,C 180,E1 -29305.443,E2 -29305.443} C_VEL
LIN {X 0,Y 80.717,Z 529.037,A -85,B 0,C 180,E1 -29310.538,E2 -29310.538} C_VEL
LIN {X 0,Y 90.903,Z 521.81,A -85,B 0,C 180,E1 -29315.288,E2 -29315.288} C_VEL
LIN {X 0,Y 100.121,Z 514.135,A -85,B 0,C 180,E1 -29318.445,E2 -29318.445} C_VEL
LIN {X 0,Y 108.583,Z 505.748,A -85,B 0,C 180,E1 -29320.96,E2 -29320.96} C_VEL
LIN {X 0,Y 117.468,Z 495.246,A -85,B 0,C 180,E1 -29323.186,E2 -29323.186} C_VEL
LIN {X 0,Y 125.616,Z 483.626,A -85,B 0,C 180,E1 -29324.816,E2 -29324.816} C_VEL
LIN {X 0,Y 132.18,Z 472.114,A -85,B 0,C 180,E1 -29326.009,E2 -29326.009} C_VEL
LIN {X 0,Y 137.895,Z 459.622,A -85,B 0,C 180,E1 -29326.889,E2 -29326.889} C_VEL
LIN {X 0,Y 142.454,Z 446.392,A -85,B 0,C 180,E1 -29327.578,E2 -29327.578} C_VEL
LIN {X 0,Y 145.757,Z 432.539,A -85,B 0,C 180,E1 -29328.052,E2 -29328.052} C_VEL
LIN {X 0,Y 148.234,Z 414.553,A -85,B 0,C 180,E1 -29328.44,E2 -29328.44} C_VEL
LIN {X 0,Y 148.352,Z 413.124,A -85,B 0,C 180,E1 -29328.558,E2 -29328.558} C_VEL
LIN {X 0,Y 147.354,Z 409.341,A -85,B 0,C 180,E1 -29331.775,E2 -29331.775} C_VEL
LIN {X 0,Y 146.578,Z 406.458,A -85,B 0,C 180,E1 -29335.618,E2 -29335.618} C_VEL
LIN {X 0,Y 146.248,Z 405.129,A -85,B 0,C 180,E1 -29340.001,E2 -29340.001} C_VEL
LIN {X 0,Y 146.321,Z 406.292,A -85,B 0,C 180,E1 -29343.357,E2 -29343.357} C_VEL
LIN {X 0,Y 146.729,Z 408.322,A -85,B 0,C 180,E1 -29346.49,E2 -29346.49} C_VEL
LIN {X 0,Y 147.461,Z 411.57,A -85,B 0,C 180,E1 -29349.69,E2 -29349.69} C_VEL
LIN {X 0,Y 148.189,Z 414.699,A -85,B 0,C 180,E1 -29352.003,E2 -29352.003} C_VEL
LIN {X 0,Y 148.138,Z 415.237,A -85,B 0,C 180,E1 -29352.033,E2 -29352.033} C_VEL
LIN {X 0,Y 147.604,Z 419.157,A -85,B 0,C 180,E1 -29351.941,E2 -29351.941} C_VEL
LIN {X 0,Y 146.301,Z 425.309,A -85,B 0,C 180,E1 -29350.965,E2 -29350.965} C_VEL
LIN {X 0,Y 144.793,Z 431.426,A -85,B 0,C 180,E1 -29349.936,E2 -29349.936} C_VEL
LIN {X 0,Y 143.879,Z 435.304,A -85,B 0,C 180,E1 -29349.783,E2 -29349.783} C_VEL
LIN {X 0,Y 140.078,Z 449.353,A -85,B 0,C 180,E1 -29350.237,E2 -29350.237} C_VEL
LIN {X 0,Y 135.114,Z 462.512,A -85,B 0,C 180,E1 -29350.956,E2 -29350.956} C_VEL
LIN {X 0,Y 129.267,Z 474.426,A -85,B 0,C 180,E1 -29351.871,E2 -29351.871} C_VEL
LIN {X 0,Y 122.609,Z 485.299,A -85,B 0,C 180,E1 -29352.985,E2 -29352.985} C_VEL
LIN {X 0,Y 114.375,Z 496.289,A -85,B 0,C 180,E1 -29354.585,E2 -29354.585} C_VEL
LIN {X 0,Y 106.205,Z 505.338,A -85,B 0,C 180,E1 -29356.36,E2 -29356.36} C_VEL
LIN {X 0,Y 96.525,Z 514.275,A -85,B 0,C 180,E1 -29358.823,E2 -29358.823} C_VEL
LIN {X 0,Y 87.12,Z 521.581,A -85,B 0,C 180,E1 -29361.922,E2 -29361.922} C_VEL
LIN {X 0,Y 78.001,Z 527.538,A -85,B 0,C 180,E1 -29365.71,E2 -29365.71} C_VEL
LIN {X 0,Y 69.738,Z 532.145,A -85,B 0,C 180,E1 -29370.26,E2 -29370.26} C_VEL
LIN {X 0,Y 61.335,Z 536.136,A -85,B 0,C 180,E1 -29376.671,E2 -29376.671} C_VEL
LIN {X 0,Y 51.934,Z 539.721,A -85,B 0,C 180,E1 -29387.42,E2 -29387.42} C_VEL
LIN {X 0,Y 45.102,Z 541.8,A -85,B 0,C 180,E1 -29402.13,E2 -29402.13} C_VEL
LIN {X 0,Y 41.641,Z 542.411,A -85,B 0,C 180,E1 -29420.283,E2 -29420.283} C_VEL
LIN {X 0,Y 41.411,Z 542.17,A -85,B 0,C 180,E1 -29429.999,E2 -29429.999} C_VEL
LIN {X 0,Y 42.103,Z 541.579,A -85,B 0,C 180,E1 -29439.608,E2 -29439.608} C_VEL
LIN {X 0,Y 46.179,Z 539.333,A -85,B 0,C 180,E1 -29457.165,E2 -29457.165} C_VEL
LIN {X 0,Y 53.492,Z 535.582,A -85,B 0,C 180,E1 -29471.064,E2 -29471.064} C_VEL
LIN {X 0,Y 60.483,Z 531.651,A -85,B 0,C 180,E1 -29479.049,E2 -29479.049} C_VEL
LIN {X 0,Y 68.409,Z 526.682,A -85,B 0,C 180,E1 -29485.271,E2 -29485.271} C_VEL
LIN {X 0,Y 78.367,Z 519.441,A -85,B 0,C 180,E1 -29490.97,E2 -29490.97} C_VEL
LIN {X 0,Y 87.417,Z 511.684,A -85,B 0,C 180,E1 -29494.747,E2 -29494.747} C_VEL
LIN {X 0,Y 96.713,Z 502.168,A -85,B 0,C 180,E1 -29497.896,E2 -29497.896} C_VEL
LIN {X 0,Y 103.875,Z 493.566,A -85,B 0,C 180,E1 -29499.84,E2 -29499.84} C_VEL
LIN {X 0,Y 111.134,Z 483.209,A -85,B 0,C 180,E1 -29501.544,E2 -29501.544} C_VEL
LIN {X 0,Y 117.645,Z 471.902,A -85,B 0,C 180,E1 -29502.903,E2 -29502.903} C_VEL
LIN {X 0,Y 123.386,Z 459.408,A -85,B 0,C 180,E1 -29503.981,E2 -29503.981} C_VEL
LIN {X 0,Y 127.318,Z 448.314,A -85,B 0,C 180,E1 -29504.674,E2 -29504.674} C_VEL
LIN {X 0,Y 130.813,Z 434.862,A -85,B 0,C 180,E1 -29505.249,E2 -29505.249} C_VEL
LIN {X 0,Y 133.022,Z 420.7,A -85,B 0,C 180,E1 -29505.628,E2 -29505.628} C_VEL
LIN {X 0,Y 134.439,Z 407.765,A -85,B 0,C 180,E1 -29506.006,E2 -29506.006} C_VEL
LIN {X 0,Y 133.505,Z 403.397,A -85,B 0,C 180,E1 -29509.573,E2 -29509.573} C_VEL
LIN {X 0,Y 132.92,Z 400.596,A -85,B 0,C 180,E1 -29513.167,E2 -29513.167} C_VEL
LIN {X 0,Y 132.7,Z 399.079,A -85,B 0,C 180,E1 -29516.963,E2 -29516.963} C_VEL
LIN {X 0,Y 132.804,Z 399.216,A -85,B 0,C 180,E1 -29520.378,E2 -29520.378} C_VEL
LIN {X 0,Y 133.174,Z 400.526,A -85,B 0,C 180,E1 -29523.537,E2 -29523.537} C_VEL
LIN {X 0,Y 134.054,Z 403.888,A -85,B 0,C 180,E1 -29527.613,E2 -29527.613} C_VEL
LIN {X 0,Y 134.631,Z 406.326,A -85,B 0,C 180,E1 -29529.589,E2 -29529.589} C_VEL
LIN {X 0,Y 131.556,Z 430.952,A -85,B 0,C 180,E1 -29530.239,E2 -29530.239} C_VEL
LIN {X 0,Y 128.313,Z 445.112,A -85,B 0,C 180,E1 -29530.747,E2 -29530.747} C_VEL
LIN {X 0,Y 124.105,Z 457.717,A -85,B 0,C 180,E1 -29531.369,E2 -29531.369} C_VEL
LIN {X 0,Y 118.704,Z 470.122,A -85,B 0,C 180,E1 -29532.346,E2 -29532.346} C_VEL
LIN {X 0,Y 112.074,Z 482.046,A -85,B 0,C 180,E1 -29533.599,E2 -29533.599} C_VEL
LIN {X 0,Y 104.725,Z 492.905,A -85,B 0,C 180,E1 -29535.274,E2 -29535.274} C_VEL
LIN {X 0,Y 95.871,Z 503.721,A -85,B 0,C 180,E1 -29537.642,E2 -29537.642} C_VEL
LIN {X 0,Y 86.386,Z 513.336,A -85,B 0,C 180,E1 -29540.679,E2 -29540.679} C_VEL
LIN {X 0,Y 77.23,Z 521.181,A -85,B 0,C 180,E1 -29544.497,E2 -29544.497} C_VEL
LIN {X 0,Y 68.532,Z 527.614,A -85,B 0,C 180,E1 -29549.348,E2 -29549.348} C_VEL
LIN {X 0,Y 60.478,Z 532.843,A -85,B 0,C 180,E1 -29555.567,E2 -29555.567} C_VEL
LIN {X 0,Y 53.393,Z 537.013,A -85,B 0,C 180,E1 -29563.62,E2 -29563.62} C_VEL
LIN {X 0,Y 47.464,Z 540.226,A -85,B 0,C 180,E1 -29573.682,E2 -29573.682} C_VEL
LIN {X 0,Y 42.409,Z 543.145,A -85,B 0,C 180,E1 -29590.645,E2 -29590.645} C_VEL
LIN {X 0,Y 41.36,Z 544.048,A -85,B 0,C 180,E1 -29600.217,E2 -29600.217} C_VEL
LIN {X 0,Y 41.273,Z 544.582,A -85,B 0,C 180,E1 -29610.001,E2 -29610.001} C_VEL
LIN {X 0,Y 41.377,Z 544.71,A -85,B 0,C 180,E1 -29619.78,E2 -29619.78} C_VEL
LIN {X 0,Y 44.535,Z 543.866,A -85,B 0,C 180,E1 -29638.257,E2 -29638.257} C_VEL
LIN {X 0,Y 51.364,Z 541.584,A -85,B 0,C 180,E1 -29653.167,E2 -29653.167} C_VEL
LIN {X 0,Y 60.653,Z 537.802,A -85,B 0,C 180,E1 -29664.203,E2 -29664.203} C_VEL
LIN {X 0,Y 68.739,Z 533.848,A -85,B 0,C 180,E1 -29670.348,E2 -29670.348} C_VEL
LIN {X 0,Y 77.447,Z 528.891,A -85,B 0,C 180,E1 -29675.154,E2 -29675.154} C_VEL
LIN {X 0,Y 88.162,Z 521.674,A -85,B 0,C 180,E1 -29679.498,E2 -29679.498} C_VEL
LIN {X 0,Y 97.727,Z 514.007,A -85,B 0,C 180,E1 -29682.336,E2 -29682.336} C_VEL
LIN {X 0,Y 107.359,Z 504.679,A -85,B 0,C 180,E1 -29684.821,E2 -29684.821} C_VEL
LIN {X 0,Y 116.444,Z 494.062,A -85,B 0,C 180,E1 -29686.709,E2 -29686.709} C_VEL
LIN {X 0,Y 124.785,Z 482.227,A -85,B 0,C 180,E1 -29688.113,E2 -29688.113} C_VEL
LIN {X 0,Y 131.493,Z 470.424,A -85,B 0,C 180,E1 -29689.138,E2 -29689.138} C_VEL
LIN {X 0,Y 137.061,Z 458.008,A -85,B 0,C 180,E1 -29689.877,E2 -29689.877} C_VEL
LIN {X 0,Y 141.595,Z 444.493,A -85,B 0,C 180,E1 -29690.448,E2 -29690.448} C_VEL
LIN {X 0,Y 144.679,Z 431.182,A -85,B 0,C 180,E1 -29690.83,E2 -29690.83} C_VEL
LIN {X 0,Y 146.572,Z 417.632,A -85,B 0,C 180,E1 -29691.12,E2 -29691.12} C_VEL
LIN {X 0,Y 145.928,Z 414.957,A -85,B 0,C 180,E1 -29693.953,E2 -29693.953} C_VEL
LIN {X 0,Y 145.614,Z 413.336,A -85,B 0,C 180,E1 -29696.196,E2 -29696.196} C_VEL
LIN {X 0,Y 145.379,Z 412.206,A -85,B 0,C 180,E1 -29700.001,E2 -29700.001} C_VEL
LIN {X 0,Y 145.42,Z 413.358,A -85,B 0,C 180,E1 -29703.118,E2 -29703.118} C_VEL
LIN {X 0,Y 145.691,Z 415.081,A -85,B 0,C 180,E1 -29705.711,E2 -29705.711} C_VEL
LIN {X 0,Y 146.299,Z 418.304,A -85,B 0,C 180,E1 -29708.896,E2 -29708.896} C_VEL
LIN {X 0,Y 146.419,Z 418.927,A -85,B 0,C 180,E1 -29709.388,E2 -29709.388} C_VEL
LIN {X 0,Y 144.181,Z 433.866,A -85,B 0,C 180,E1 -29709.736,E2 -29709.736} C_VEL
LIN {X 0,Y 143.879,Z 435.304,A -85,B 0,C 180,E1 -29709.783,E2 -29709.783} C_VEL
LIN {X 0,Y 142.894,Z 439.152,A -85,B 0,C 180,E1 -29709.636,E2 -29709.636} C_VEL
LIN {X 0,Y 140.824,Z 445.155,A -85,B 0,C 180,E1 -29708.666,E2 -29708.666} C_VEL
LIN {X 0,Y 138.558,Z 451.073,A -85,B 0,C 180,E1 -29707.687,E2 -29707.687} C_VEL
LIN {X 0,Y 137.134,Z 454.783,A -85,B 0,C 180,E1 -29707.596,E2 -29707.596} C_VEL
LIN {X 0,Y 131.389,Z 468.057,A -85,B 0,C 180,E1 -29708.292,E2 -29708.292} C_VEL
LIN {X 0,Y 124.592,Z 480.251,A -85,B 0,C 180,E1 -29709.204,E2 -29709.204} C_VEL
LIN {X 0,Y 116.845,Z 491.375,A -85,B 0,C 180,E1 -29710.397,E2 -29710.397} C_VEL
LIN {X 0,Y 107.771,Z 502.023,A -85,B 0,C 180,E1 -29711.993,E2 -29711.993} C_VEL
LIN {X 0,Y 97.77,Z 511.637,A -85,B 0,C 180,E1 -29713.973,E2 -29713.973} C_VEL
LIN {X 0,Y 87.959,Z 519.47,A -85,B 0,C 180,E1 -29716.505,E2 -29716.505} C_VEL
LIN {X 0,Y 78.334,Z 525.857,A -85,B 0,C 180,E1 -29719.604,E2 -29719.604} C_VEL
LIN {X 0,Y 69.004,Z 531.028,A -85,B 0,C 180,E1 -29723.562,E2 -29723.562} C_VEL
LIN {X 0,Y 60.185,Z 535.134,A -85,B 0,C 180,E1 -29728.861,E2 -29728.861} C_VEL
LIN {X 0,Y 51.96,Z 538.291,A -85,B 0,C 180,E1 -29735.753,E2 -29735.753} C_VEL
LIN {X 0,Y 42.562,Z 541.124,A -85,B 0,C 180,E1 -29748.663,E2 -29748.663} C_VEL
LIN {X 0,Y 36.247,Z 542.488,A -85,B 0,C 180,E1 -29767.183,E2 -29767.183} C_VEL
LIN {X 0,Y 34.312,Z 542.377,A -85,B 0,C 180,E1 -29789.999,E2 -29789.999} C_VEL
LIN {X 0,Y 35.134,Z 541.792,A -85,B 0,C 180,E1 -29801.538,E2 -29801.538} C_VEL
LIN {X 0,Y 40.009,Z 539.557,A -85,B 0,C 180,E1 -29821.8,E2 -29821.8} C_VEL
LIN {X 0,Y 48.362,Z 535.824,A -85,B 0,C 180,E1 -29836.6,E2 -29836.6} C_VEL
LIN {X 0,Y 56.096,Z 531.903,A -85,B 0,C 180,E1 -29844.522,E2 -29844.522} C_VEL
LIN {X 0,Y 64.639,Z 526.951,A -85,B 0,C 180,E1 -29850.435,E2 -29850.435} C_VEL
LIN {X 0,Y 75.179,Z 519.736,A -85,B 0,C 180,E1 -29855.706,E2 -29855.706} C_VEL
LIN {X 0,Y 84.642,Z 512.012,A -85,B 0,C 180,E1 -29859.081,E2 -29859.081} C_VEL
LIN {X 0,Y 94.281,Z 502.529,A -85,B 0,C 180,E1 -29861.88,E2 -29861.88} C_VEL
LIN {X 0,Y 101.655,Z 493.97,A -85,B 0,C 180,E1 -29863.585,E2 -29863.585} C_VEL
LIN {X 0,Y 109.102,Z 483.67,A -85,B 0,C 180,E1 -29865.067,E2 -29865.067} C_VEL
LIN {X 0,Y 115.761,Z 472.443,A -85,B 0,C 180,E1 -29866.255,E2 -29866.255} C_VEL
LIN {X 0,Y 121.625,Z 460.061,A -85,B 0,C 180,E1 -29867.183,E2 -29867.183} C_VEL
LIN {X 0,Y 126.081,Z 447.773,A -85,B 0,C 180,E1 -29867.85,E2 -29867.85} C_VEL
LIN {X 0,Y 129.612,Z 434.12,A -85,B 0,C 180,E1 -29868.346,E2 -29868.346} C_VEL
LIN {X 0,Y 131.933,Z 418.795,A -85,B 0,C 180,E1 -29868.672,E2 -29868.672} C_VEL
LIN {X 0,Y 132.7,Z 411.942,A -85,B 0,C 180,E1 -29868.877,E2 -29868.877} C_VEL
LIN {X 0,Y 132.232,Z 409.353,A -85,B 0,C 180,E1 -29871.402,E2 -29871.402} C_VEL
LIN {X 0,Y 131.956,Z 407.441,A -85,B 0,C 180,E1 -29873.884,E2 -29873.884} C_VEL
LIN {X 0,Y 131.827,Z 406.189,A -85,B 0,C 180,E1 -29876.943,E2 -29876.943} C_VEL
LIN {X 0,Y 131.96,Z 406.435,A -85,B 0,C 180,E1 -29880.762,E2 -29880.762} C_VEL
LIN {X 0,Y 132.177,Z 407.41,A -85,B 0,C 180,E1 -29882.856,E2 -29882.856} C_VEL
LIN {X 0,Y 132.877,Z 410.631,A -85,B 0,C 180,E1 -29886.734,E2 -29886.734} C_VEL
LIN {X 0,Y 130.265,Z 430.673,A -85,B 0,C 180,E1 -29887.185,E2 -29887.185} C_VEL
LIN {X 0,Y 126.934,Z 445.018,A -85,B 0,C 180,E1 -29887.621,E2 -29887.621} C_VEL
LIN {X 0,Y 122.456,Z 458.163,A -85,B 0,C 180,E1 -29888.168,E2 -29888.168} C_VEL
LIN {X 0,Y 116.539,Z 471.189,A -85,B 0,C 180,E1 -29889.072,E2 -29889.072} C_VEL
LIN {X 0,Y 109.768,Z 482.883,A -85,B 0,C 180,E1 -29890.142,E2 -29890.142} C_VEL
LIN {X 0,Y 102.238,Z 493.576,A -85,B 0,C 180,E1 -29891.608,E2 -29891.608} C_VEL
LIN {X 0,Y 93.959,Z 503.359,A -85,B 0,C 180,E1 -29893.503,E2 -29893.503} C_VEL
LIN {X 0,Y 84.126,Z 513.006,A -85,B 0,C 180,E1 -29896.116,E2 -29896.116} C_VEL
LIN {X 0,Y 74.546,Z 520.884,A -85,B 0,C 180,E1 -29899.481,E2 -29899.481} C_VEL
LIN {X 0,Y 65.319,Z 527.336,A -85,B 0,C 180,E1 -29903.86,E2 -29903.86} C_VEL
LIN {X 0,Y 56.156,Z 532.849,A -85,B 0,C 180,E1 -29910.038,E2 -29910.038} C_VEL
LIN {X 0,Y 48.725,Z 536.766,A -85,B 0,C 180,E1 -29917.506,E2 -29917.506} C_VEL
LIN {X 0,Y 41.928,Z 539.994,A -85,B 0,C 180,E1 -29927.897,E2 -29927.897} C_VEL
LIN {X 0,Y 35.755,Z 542.925,A -85,B 0,C 180,E1 -29946.853,E2 -29946.853} C_VEL
LIN {X 0,Y 34.359,Z 543.834,A -85,B 0,C 180,E1 -29958.198,E2 -29958.198} C_VEL
LIN {X 0,Y 34.157,Z 544.375,A -85,B 0,C 180,E1 -29970.001,E2 -29970.001} C_VEL
LIN {X 0,Y 34.378,Z 544.513,A -85,B 0,C 180,E1 -29981.797,E2 -29981.797} C_VEL
LIN {X 0,Y 38.394,Z 543.68,A -85,B 0,C 180,E1 -30003.308,E2 -30003.308} C_VEL
LIN {X 0,Y 46.416,Z 541.408,A -85,B 0,C 180,E1 -30019.206,E2 -30019.206} C_VEL
LIN {X 0,Y 54.045,Z 538.718,A -85,B 0,C 180,E1 -30027.698,E2 -30027.698} C_VEL
LIN {X 0,Y 62.522,Z 535.132,A -85,B 0,C 180,E1 -30034.06,E2 -30034.06} C_VEL
LIN {X 0,Y 71.602,Z 530.539,A -85,B 0,C 180,E1 -30038.819,E2 -30038.819} C_VEL
LIN {X 0,Y 82.69,Z 523.783,A -85,B 0,C 180,E1 -30042.969,E2 -30042.969} C_VEL
LIN {X 0,Y 92.497,Z 516.599,A -85,B 0,C 180,E1 -30045.638,E2 -30045.638} C_VEL
LIN {X 0,Y 102.13,Z 508.128,A -85,B 0,C 180,E1 -30047.801,E2 -30047.801} C_VEL
LIN {X 0,Y 110.797,Z 499.014,A -85,B 0,C 180,E1 -30049.473,E2 -30049.473} C_VEL
LIN {X 0,Y 119.259,Z 488.354,A -85,B 0,C 180,E1 -30050.776,E2 -30050.776} C_VEL
LIN {X 0,Y 126.923,Z 476.542,A -85,B 0,C 180,E1 -30051.796,E2 -30051.796} C_VEL
LIN {X 0,Y 132.919,Z 465.052,A -85,B 0,C 180,E1 -30052.472,E2 -30052.472} C_VEL
LIN {X 0,Y 138.274,Z 451.749,A -85,B 0,C 180,E1 -30053.064,E2 -30053.064} C_VEL
LIN {X 0,Y 142.206,Z 438.204,A -85,B 0,C 180,E1 -30053.46,E2 -30053.46} C_VEL
LIN {X 0,Y 144.799,Z 424.212,A -85,B 0,C 180,E1 -30053.743,E2 -30053.743} C_VEL
LIN {X 0,Y 145.026,Z 422.315,A -85,B 0,C 180,E1 -30053.892,E2 -30053.892} C_VEL
LIN {X 0,Y 144.653,Z 420.172,A -85,B 0,C 180,E1 -30056.868,E2 -30056.868} C_VEL
LIN {X 0,Y 144.51,Z 419.285,A -85,B 0,C 180,E1 -30060.001,E2 -30060.001} C_VEL
LIN {X 0,Y 144.535,Z 420.578,A -85,B 0,C 180,E1 -30063.137,E2 -30063.137} C_VEL
LIN {X 0,Y 144.71,Z 422.123,A -85,B 0,C 180,E1 -30065.226,E2 -30065.226} C_VEL
LIN {X 0,Y 144.896,Z 423.472,A -85,B 0,C 180,E1 -30066.7,E2 -30066.7} C_VEL
LIN {X 0,Y 142.306,Z 437.764,A -85,B 0,C 180,E1 -30067.052,E2 -30067.052} C_VEL
LIN {X 0,Y 138.224,Z 451.801,A -85,B 0,C 180,E1 -30067.449,E2 -30067.449} C_VEL
LIN {X 0,Y 137.134,Z 454.783,A -85,B 0,C 180,E1 -30067.596,E2 -30067.596} C_VEL
LIN {X 0,Y 134.885,Z 460.301,A -85,B 0,C 180,E1 -30067.631,E2 -30067.631} C_VEL
LIN {X 0,Y 130.513,Z 468.998,A -85,B 0,C 180,E1 -30066.886,E2 -30066.886} C_VEL
LIN {X 0,Y 125.546,Z 477.399,A -85,B 0,C 180,E1 -30066.092,E2 -30066.092} C_VEL
LIN {X 0,Y 122.328,Z 482.351,A -85,B 0,C 180,E1 -30066.106,E2 -30066.106} C_VEL
LIN {X 0,Y 114.309,Z 493.309,A -85,B 0,C 180,E1 -30067.137,E2 -30067.137} C_VEL
LIN {X 0,Y 104.816,Z 503.916,A -85,B 0,C 180,E1 -30068.513,E2 -30068.513} C_VEL
LIN {X 0,Y 94.613,Z 513.179,A -85,B 0,C 180,E1 -30070.193,E2 -30070.193} C_VEL
LIN {X 0,Y 84.536,Z 520.74,A -85,B 0,C 180,E1 -30072.357,E2 -30072.357} C_VEL
LIN {X 0,Y 72.96,Z 527.828,A -85,B 0,C 180,E1 -30075.581,E2 -30075.581} C_VEL
LIN {X 0,Y 62.389,Z 533.064,A -85,B 0,C 180,E1 -30079.754,E2 -30079.754} C_VEL
LIN {X 0,Y 54.034,Z 536.465,A -85,B 0,C 180,E1 -30084.432,E2 -30084.432} C_VEL
LIN {X 0,Y 42.548,Z 540.071,A -85,B 0,C 180,E1 -30094.323,E2 -30094.323} C_VEL
LIN {X 0,Y 33.189,Z 542.172,A -85,B 0,C 180,E1 -30110.559,E2 -30110.559} C_VEL
LIN {X 0,Y 29.83,Z 542.681,A -85,B 0,C 180,E1 -30121.887,E2 -30121.887} C_VEL
LIN {X 0,Y 27.228,Z 542.584,A -85,B 0,C 180,E1 -30149.999,E2 -30149.999} C_VEL
LIN {X 0,Y 28.239,Z 542.004,A -85,B 0,C 180,E1 -30164.41,E2 -30164.41} C_VEL
LIN {X 0,Y 34.184,Z 539.782,A -85,B 0,C 180,E1 -30188.08,E2 -30188.08} C_VEL
LIN {X 0,Y 43.793,Z 536.065,A -85,B 0,C 180,E1 -30203.358,E2 -30203.358} C_VEL
LIN {X 0,Y 52.306,Z 532.154,A -85,B 0,C 180,E1 -30210.85,E2 -30210.85} C_VEL
LIN {X 0,Y 61.446,Z 527.221,A -85,B 0,C 180,E1 -30216.204,E2 -30216.204} C_VEL
LIN {X 0,Y 72.549,Z 520.028,A -85,B 0,C 180,E1 -30220.819,E2 -30220.819} C_VEL
LIN {X 0,Y 82.382,Z 512.336,A -85,B 0,C 180,E1 -30223.68,E2 -30223.68} C_VEL
LIN {X 0,Y 92.327,Z 502.89,A -85,B 0,C 180,E1 -30226.053,E2 -30226.053} C_VEL
LIN {X 0,Y 99.887,Z 494.374,A -85,B 0,C 180,E1 -30227.479,E2 -30227.479} C_VEL
LIN {X 0,Y 106.347,Z 485.816,A -85,B 0,C 180,E1 -30228.583,E2 -30228.583} C_VEL
LIN {X 0,Y 113.439,Z 474.555,A -85,B 0,C 180,E1 -30229.578,E2 -30229.578} C_VEL
LIN {X 0,Y 119.404,Z 462.692,A -85,B 0,C 180,E1 -30230.356,E2 -30230.356} C_VEL
LIN {X 0,Y 123.978,Z 451.044,A -85,B 0,C 180,E1 -30230.937,E2 -30230.937} C_VEL
LIN {X 0,Y 127.948,Z 437.159,A -85,B 0,C 180,E1 -30231.377,E2 -30231.377} C_VEL
LIN {X 0,Y 130.371,Z 423.789,A -85,B 0,C 180,E1 -30231.668,E2 -30231.668} C_VEL
LIN {X 0,Y 131.265,Z 416.444,A -85,B 0,C 180,E1 -30231.809,E2 -30231.809} C_VEL
LIN {X 0,Y 131.017,Z 414.258,A -85,B 0,C 180,E1 -30234.612,E2 -30234.612} C_VEL
LIN {X 0,Y 130.954,Z 413.31,A -85,B 0,C 180,E1 -30236.923,E2 -30236.923} C_VEL
LIN {X 0,Y 131.086,Z 413.551,A -85,B 0,C 180,E1 -30240.767,E2 -30240.767} C_VEL
LIN {X 0,Y 131.239,Z 414.593,A -85,B 0,C 180,E1 -30242.589,E2 -30242.589} C_VEL
LIN {X 0,Y 131.38,Z 415.495,A -85,B 0,C 180,E1 -30243.76,E2 -30243.76} C_VEL
LIN {X 0,Y 128.999,Z 432.264,A -85,B 0,C 180,E1 -30244.119,E2 -30244.119} C_VEL
LIN {X 0,Y 125.591,Z 446.162,A -85,B 0,C 180,E1 -30244.477,E2 -30244.477} C_VEL
LIN {X 0,Y 121.44,Z 457.984,A -85,B 0,C 180,E1 -30244.877,E2 -30244.877} C_VEL
LIN {X 0,Y 115.631,Z 470.65,A -85,B 0,C 180,E1 -30245.588,E2 -30245.588} C_VEL
LIN {X 0,Y 108.743,Z 482.422,A -85,B 0,C 180,E1 -30246.456,E2 -30246.456} C_VEL
LIN {X 0,Y 101.042,Z 493.169,A -85,B 0,C 180,E1 -30247.634,E2 -30247.634} C_VEL
LIN {X 0,Y 92.554,Z 502.997,A -85,B 0,C 180,E1 -30249.205,E2 -30249.205} C_VEL
LIN {X 0,Y 82.432,Z 512.677,A -85,B 0,C 180,E1 -30251.348,E2 -30251.348} C_VEL
LIN {X 0,Y 72.466,Z 520.583,A -85,B 0,C 180,E1 -30254.116,E2 -30254.116} C_VEL
LIN {X 0,Y 62.767,Z 527.056,A -85,B 0,C 180,E1 -30257.876,E2 -30257.876} C_VEL
LIN {X 0,Y 52.08,Z 533.022,A -85,B 0,C 180,E1 -30263.878,E2 -30263.878} C_VEL
LIN {X 0,Y 42.005,Z 537.713,A -85,B 0,C 180,E1 -30273.224,E2 -30273.224} C_VEL
LIN {X 0,Y 32.594,Z 541.421,A -85,B 0,C 180,E1 -30289.696,E2 -30289.696} C_VEL
LIN {X 0,Y 27.411,Z 543.62,A -85,B 0,C 180,E1 -30315.145,E2 -30315.145} C_VEL
LIN {X 0,Y 27.046,Z 544.169,A -85,B 0,C 180,E1 -30330.001,E2 -30330.001} C_VEL
LIN {X 0,Y 27.454,Z 544.315,A -85,B 0,C 180,E1 -30344.833,E2 -30344.833} C_VEL
LIN {X 0,Y 32.648,Z 543.493,A -85,B 0,C 180,E1 -30370.225,E2 -30370.225} C_VEL
LIN {X 0,Y 42.094,Z 541.232,A -85,B 0,C 180,E1 -30386.595,E2 -30386.595} C_VEL
LIN {X 0,Y 50.574,Z 538.551,A -85,B 0,C 180,E1 -30394.59,E2 -30394.59} C_VEL
LIN {X 0,Y 59.741,Z 534.976,A -85,B 0,C 180,E1 -30400.24,E2 -30400.24} C_VEL
LIN {X 0,Y 69.339,Z 530.388,A -85,B 0,C 180,E1 -30404.341,E2 -30404.341} C_VEL
LIN {X 0,Y 80.889,Z 523.646,A -85,B 0,C 180,E1 -30407.807,E2 -30407.807} C_VEL
LIN {X 0,Y 90.992,Z 516.471,A -85,B 0,C 180,E1 -30409.985,E2 -30409.985} C_VEL
LIN {X 0,Y 101.579,Z 507.321,A -85,B 0,C 180,E1 -30411.885,E2 -30411.885} C_VEL
LIN {X 0,Y 111.436,Z 496.945,A -85,B 0,C 180,E1 -30413.362,E2 -30413.362} C_VEL
LIN {X 0,Y 120.056,Z 485.884,A -85,B 0,C 180,E1 -30414.357,E2 -30414.357} C_VEL
LIN {X 0,Y 126.97,Z 474.967,A -85,B 0,C 180,E1 -30415.08,E2 -30415.08} C_VEL
LIN {X 0,Y 133.042,Z 463.037,A -85,B 0,C 180,E1 -30415.61,E2 -30415.61} C_VEL
LIN {X 0,Y 138.34,Z 449.409,A -85,B 0,C 180,E1 -30416.06,E2 -30416.06} C_VEL
LIN {X 0,Y 142.204,Z 435.399,A -85,B 0,C 180,E1 -30416.371,E2 -30416.371} C_VEL
LIN {X 0,Y 143.679,Z 427.522,A -85,B 0,C 180,E1 -30416.565,E2 -30416.565} C_VEL
LIN {X 0,Y 143.552,Z 426.493,A -85,B 0,C 180,E1 -30419.3,E2 -30419.3} C_VEL
LIN {X 0,Y 143.521,Z 426.696,A -85,B 0,C 180,E1 -30421.141,E2 -30421.141} C_VEL
LIN {X 0,Y 143.552,Z 428.391,A -85,B 0,C 180,E1 -30423.945,E2 -30423.945} C_VEL
LIN {X 0,Y 140.725,Z 441.453,A -85,B 0,C 180,E1 -30424.263,E2 -30424.263} C_VEL
LIN {X 0,Y 136.55,Z 454.43,A -85,B 0,C 180,E1 -30424.609,E2 -30424.609} C_VEL
LIN {X 0,Y 131.417,Z 466.393,A -85,B 0,C 180,E1 -30425.113,E2 -30425.113} C_VEL
LIN {X 0,Y 124.518,Z 478.942,A -85,B 0,C 180,E1 -30425.863,E2 -30425.863} C_VEL
LIN {X 0,Y 122.328,Z 482.351,A -85,B 0,C 180,E1 -30426.106,E2 -30426.106} C_VEL
LIN {X 0,Y 118.903,Z 487.227,A -85,B 0,C 180,E1 -30426.167,E2 -30426.167} C_VEL
LIN {X 0,Y 112.718,Z 494.846,A -85,B 0,C 180,E1 -30425.477,E2 -30425.477} C_VEL
LIN {X 0,Y 106.035,Z 502.019,A -85,B 0,C 180,E1 -30424.766,E2 -30424.766} C_VEL
LIN {X 0,Y 101.805,Z 506.126,A -85,B 0,C 180,E1 -30424.887,E2 -30424.887} C_VEL
LIN {X 0,Y 91.887,Z 514.656,A -85,B 0,C 180,E1 -30426.126,E2 -30426.126} C_VEL
LIN {X 0,Y 81.592,Z 521.987,A -85,B 0,C 180,E1 -30427.882,E2 -30427.882} C_VEL
LIN {X 0,Y 71.377,Z 527.973,A -85,B 0,C 180,E1 -30430.064,E2 -30430.064} C_VEL
LIN {X 0,Y 59.533,Z 533.569,A -85,B 0,C 180,E1 -30433.659,E2 -30433.659} C_VEL
LIN {X 0,Y 48.293,Z 537.685,A -85,B 0,C 180,E1 -30438.927,E2 -30438.927} C_VEL
LIN {X 0,Y 38.981,Z 540.247,A -85,B 0,C 180,E1 -30445.65,E2 -30445.65} C_VEL
LIN {X 0,Y 28.043,Z 542.359,A -85,B 0,C 180,E1 -30461.25,E2 -30461.25} C_VEL
LIN {X 0,Y 23.783,Z 542.874,A -85,B 0,C 180,E1 -30473.77,E2 -30473.77} C_VEL
LIN {X 0,Y 20.12,Z 542.792,A -85,B 0,C 180,E1 -30509.999,E2 -30509.999} C_VEL
LIN {X 0,Y 21.443,Z 542.217,A -85,B 0,C 180,E1 -30529.131,E2 -30529.131} C_VEL
LIN {X 0,Y 28.94,Z 540.006,A -85,B 0,C 180,E1 -30556.763,E2 -30556.763} C_VEL
LIN {X 0,Y 39.971,Z 536.305,A -85,B 0,C 180,E1 -30571.537,E2 -30571.537} C_VEL
LIN {X 0,Y 49.248,Z 532.406,A -85,B 0,C 180,E1 -30578.058,E2 -30578.058} C_VEL
LIN {X 0,Y 58.941,Z 527.49,A -85,B 0,C 180,E1 -30582.531,E2 -30582.531} C_VEL
LIN {X 0,Y 70.539,Z 520.318,A -85,B 0,C 180,E1 -30586.263,E2 -30586.263} C_VEL
LIN {X 0,Y 80.681,Z 512.658,A -85,B 0,C 180,E1 -30588.506,E2 -30588.506} C_VEL
LIN {X 0,Y 90.883,Z 503.251,A -85,B 0,C 180,E1 -30590.381,E2 -30590.381} C_VEL
LIN {X 0,Y 98.596,Z 494.778,A -85,B 0,C 180,E1 -30591.492,E2 -30591.492} C_VEL
LIN {X 0,Y 106.339,Z 484.593,A -85,B 0,C 180,E1 -30592.454,E2 -30592.454} C_VEL
LIN {X 0,Y 113.24,Z 473.519,A -85,B 0,C 180,E1 -30593.211,E2 -30593.211} C_VEL
LIN {X 0,Y 119.289,Z 461.367,A -85,B 0,C 180,E1 -30593.816,E2 -30593.816} C_VEL
LIN {X 0,Y 124.047,Z 448.937,A -85,B 0,C 180,E1 -30594.262,E2 -30594.262} C_VEL
LIN {X 0,Y 127.731,Z 435.572,A -85,B 0,C 180,E1 -30594.579,E2 -30594.579} C_VEL
LIN {X 0,Y 130.028,Z 422.204,A -85,B 0,C 180,E1 -30594.796,E2 -30594.796} C_VEL
LIN {X 0,Y 130.117,Z 421.384,A -85,B 0,C 180,E1 -30594.89,E2 -30594.89} C_VEL
LIN {X 0,Y 130.075,Z 420.473,A -85,B 0,C 180,E1 -30596.902,E2 -30596.902} C_VEL
LIN {X 0,Y 130.203,Z 420.631,A -85,B 0,C 180,E1 -30600.663,E2 -30600.663} C_VEL
LIN {X 0,Y 128.741,Z 430.546,A -85,B 0,C 180,E1 -30600.956,E2 -30600.956} C_VEL
LIN {X 0,Y 125.482,Z 444.337,A -85,B 0,C 180,E1 -30601.201,E2 -30601.201} C_VEL
LIN {X 0,Y 120.82,Z 457.833,A -85,B 0,C 180,E1 -30601.541,E2 -30601.541} C_VEL
LIN {X 0,Y 115.156,Z 470.106,A -85,B 0,C 180,E1 -30602.061,E2 -30602.061} C_VEL
LIN {X 0,Y 108.173,Z 481.96,A -85,B 0,C 180,E1 -30602.702,E2 -30602.702} C_VEL
LIN {X 0,Y 100.342,Z 492.762,A -85,B 0,C 180,E1 -30603.574,E2 -30603.574} C_VEL
LIN {X 0,Y 91.683,Z 502.634,A -85,B 0,C 180,E1 -30604.799,E2 -30604.799} C_VEL
LIN {X 0,Y 81.33,Z 512.348,A -85,B 0,C 180,E1 -30606.419,E2 -30606.419} C_VEL
LIN {X 0,Y 71.058,Z 520.28,A -85,B 0,C 180,E1 -30608.494,E2 -30608.494} C_VEL
LIN {X 0,Y 60.948,Z 526.774,A -85,B 0,C 180,E1 -30611.444,E2 -30611.444} C_VEL
LIN {X 0,Y 48.887,Z 533.097,A -85,B 0,C 180,E1 -30616.707,E2 -30616.707} C_VEL
LIN {X 0,Y 38.545,Z 537.474,A -85,B 0,C 180,E1 -30624.268,E2 -30624.268} C_VEL
LIN {X 0,Y 32.772,Z 539.53,A -85,B 0,C 180,E1 -30630.932,E2 -30630.932} C_VEL
LIN {X 0,Y 23.308,Z 542.485,A -85,B 0,C 180,E1 -30652.913,E2 -30652.913} C_VEL
LIN {X 0,Y 20.608,Z 543.406,A -85,B 0,C 180,E1 -30670.061,E2 -30670.061} C_VEL
LIN {X 0,Y 19.949,Z 543.962,A -85,B 0,C 180,E1 -30690.001,E2 -30690.001} C_VEL
LIN {X 0,Y 20.645,Z 544.117,A -85,B 0,C 180,E1 -30709.903,E2 -30709.903} C_VEL
LIN {X 0,Y 23.377,Z 543.892,A -85,B 0,C 180,E1 -30726.961,E2 -30726.961} C_VEL
LIN {X 0,Y 32.801,Z 542.362,A -85,B 0,C 180,E1 -30748.987,E2 -30748.987} C_VEL
LIN {X 0,Y 44.783,Z 539.375,A -85,B 0,C 180,E1 -30760.322,E2 -30760.322} C_VEL
LIN {X 0,Y 54.414,Z 536.089,A -85,B 0,C 180,E1 -30765.621,E2 -30765.621} C_VEL
LIN {X 0,Y 64.388,Z 531.862,A -85,B 0,C 180,E1 -30769.218,E2 -30769.218} C_VEL
LIN {X 0,Y 76.26,Z 525.572,A -85,B 0,C 180,E1 -30772.177,E2 -30772.177} C_VEL
LIN {X 0,Y 88.3,Z 517.632,A -85,B 0,C 180,E1 -30774.208,E2 -30774.208} C_VEL
LIN {X 0,Y 98.679,Z 509.201,A -85,B 0,C 180,E1 -30775.62,E2 -30775.62} C_VEL
LIN {X 0,Y 107.356,Z 500.705,A -85,B 0,C 180,E1 -30776.676,E2 -30776.676} C_VEL
LIN {X 0,Y 116.073,Z 490.488,A -85,B 0,C 180,E1 -30777.473,E2 -30777.473} C_VEL
LIN {X 0,Y 123.936,Z 479.187,A -85,B 0,C 180,E1 -30778.085,E2 -30778.085} C_VEL
LIN {X 0,Y 130.06,Z 468.378,A -85,B 0,C 180,E1 -30778.502,E2 -30778.502} C_VEL
LIN {X 0,Y 135.802,Z 455.492,A -85,B 0,C 180,E1 -30778.863,E2 -30778.863} C_VEL
LIN {X 0,Y 140.352,Z 441.669,A -85,B 0,C 180,E1 -30779.127,E2 -30779.127} C_VEL
LIN {X 0,Y 142.297,Z 433.488,A -85,B 0,C 180,E1 -30779.32,E2 -30779.32} C_VEL
LIN {X 0,Y 142.242,Z 433.749,A -85,B 0,C 180,E1 -30781.042,E2 -30781.042} C_VEL
LIN {X 0,Y 142.23,Z 433.846,A -85,B 0,C 180,E1 -30781.211,E2 -30781.211} C_VEL
LIN {X 0,Y 138.966,Z 446.465,A -85,B 0,C 180,E1 -30781.45,E2 -30781.45} C_VEL
LIN {X 0,Y 134.466,Z 458.859,A -85,B 0,C 180,E1 -30781.763,E2 -30781.763} C_VEL
LIN {X 0,Y 128.358,Z 471.57,A -85,B 0,C 180,E1 -30782.248,E2 -30782.248} C_VEL
LIN {X 0,Y 121.378,Z 483.046,A -85,B 0,C 180,E1 -30782.82,E2 -30782.82} C_VEL
LIN {X 0,Y 112.678,Z 494.605,A -85,B 0,C 180,E1 -30783.676,E2 -30783.676} C_VEL
LIN {X 0,Y 104.002,Z 504.031,A -85,B 0,C 180,E1 -30784.641,E2 -30784.641} C_VEL
LIN {X 0,Y 101.805,Z 506.126,A -85,B 0,C 180,E1 -30784.887,E2 -30784.887} C_VEL
LIN {X 0,Y 97.394,Z 510.1,A -85,B 0,C 180,E1 -30785.02,E2 -30785.02} C_VEL
LIN {X 0,Y 89.684,Z 516.193,A -85,B 0,C 180,E1 -30784.187,E2 -30784.187} C_VEL
LIN {X 0,Y 81.596,Z 521.728,A -85,B 0,C 180,E1 -30783.27,E2 -30783.27} C_VEL
LIN {X 0,Y 76.559,Z 524.778,A -85,B 0,C 180,E1 -30783.458,E2 -30783.458} C_VEL
LIN {X 0,Y 63.558,Z 531.477,A -85,B 0,C 180,E1 -30785.634,E2 -30785.634} C_VEL
LIN {X 0,Y 53.266,Z 535.614,A -85,B 0,C 180,E1 -30788.288,E2 -30788.288} C_VEL
LIN {X 0,Y 43.116,Z 538.801,A -85,B 0,C 180,E1 -30792.039,E2 -30792.039} C_VEL
LIN {X 0,Y 30.022,Z 541.667,A -85,B 0,C 180,E1 -30800.546,E2 -30800.546} C_VEL
LIN {X 0,Y 18.526,Z 543.066,A -85,B 0,C 180,E1 -30820.647,E2 -30820.647} C_VEL
LIN {X 0,Y 14.459,Z 543.217,A -85,B 0,C 180,E1 -30840.916,E2 -30840.916} C_VEL
LIN {X 0,Y 13.014,Z 542.999,A -85,B 0,C 180,E1 -30869.998,E2 -30869.998} C_VEL
LIN {X 0,Y 14.937,Z 542.43,A -85,B 0,C 180,E1 -30898.064,E2 -30898.064} C_VEL
LIN {X 0,Y 24.628,Z 540.23,A -85,B 0,C 180,E1 -30928.877,E2 -30928.877} C_VEL
LIN {X 0,Y 37.121,Z 536.543,A -85,B 0,C 180,E1 -30941.191,E2 -30941.191} C_VEL
LIN {X 0,Y 47.059,Z 532.658,A -85,B 0,C 180,E1 -30946.097,E2 -30946.097} C_VEL
LIN {X 0,Y 57.212,Z 527.76,A -85,B 0,C 180,E1 -30949.328,E2 -30949.328} C_VEL
LIN {X 0,Y 69.2,Z 520.607,A -85,B 0,C 180,E1 -30951.967,E2 -30951.967} C_VEL
LIN {X 0,Y 79.573,Z 512.976,A -85,B 0,C 180,E1 -30953.513,E2 -30953.513} C_VEL
LIN {X 0,Y 89.97,Z 503.612,A -85,B 0,C 180,E1 -30954.834,E2 -30954.834} C_VEL
LIN {X 0,Y 97.801,Z 495.181,A -85,B 0,C 180,E1 -30955.591,E2 -30955.591} C_VEL
LIN {X 0,Y 105.641,Z 485.055,A -85,B 0,C 180,E1 -30956.27,E2 -30956.27} C_VEL
LIN {X 0,Y 112.623,Z 474.058,A -85,B 0,C 180,E1 -30956.78,E2 -30956.78} C_VEL
LIN {X 0,Y 119.174,Z 461.029,A -85,B 0,C 180,E1 -30957.229,E2 -30957.229} C_VEL
LIN {X 0,Y 123.82,Z 448.941,A -85,B 0,C 180,E1 -30957.545,E2 -30957.545} C_VEL
LIN {X 0,Y 126.603,Z 439.453,A -85,B 0,C 180,E1 -30957.699,E2 -30957.699} C_VEL
LIN {X 0,Y 126.587,Z 439.522,A -85,B 0,C 180,E1 -30957.894,E2 -30957.894} C_VEL
LIN {X 0,Y 122.717,Z 452.213,A -85,B 0,C 180,E1 -30958.087,E2 -30958.087} C_VEL
LIN {X 0,Y 117.767,Z 464.201,A -85,B 0,C 180,E1 -30958.315,E2 -30958.315} C_VEL
LIN {X 0,Y 111.595,Z 475.861,A -85,B 0,C 180,E1 -30958.711,E2 -30958.711} C_VEL
LIN {X 0,Y 103.671,Z 487.785,A -85,B 0,C 180,E1 -30959.195,E2 -30959.195} C_VEL
LIN {X 0,Y 94.597,Z 498.844,A -85,B 0,C 180,E1 -30959.999,E2 -30959.999} C_VEL
LIN {X 0,Y 84.347,Z 509.02,A -85,B 0,C 180,E1 -30960.99,E2 -30960.99} C_VEL
LIN {X 0,Y 73.847,Z 517.496,A -85,B 0,C 180,E1 -30962.203,E2 -30962.203} C_VEL
LIN {X 0,Y 61.669,Z 525.476,A -85,B 0,C 180,E1 -30964.328,E2 -30964.328} C_VEL
LIN {X 0,Y 49.624,Z 531.79,A -85,B 0,C 180,E1 -30967.544,E2 -30967.544} C_VEL
LIN {X 0,Y 39.511,Z 536.025,A -85,B 0,C 180,E1 -30971.964,E2 -30971.964} C_VEL
LIN {X 0,Y 29.731,Z 539.297,A -85,B 0,C 180,E1 -30979.003,E2 -30979.003} C_VEL
LIN {X 0,Y 18.123,Z 542.264,A -85,B 0,C 180,E1 -30999.144,E2 -30999.144} C_VEL
LIN {X 0,Y 14.13,Z 543.193,A -85,B 0,C 180,E1 -31020.174,E2 -31020.174} C_VEL
LIN {X 0,Y 12.84,Z 543.754,A -85,B 0,C 180,E1 -31050.002,E2 -31050.002} C_VEL
LIN {X 0,Y 14.164,Z 543.918,A -85,B 0,C 180,E1 -31079.75,E2 -31079.75} C_VEL
LIN {X 0,Y 23.607,Z 543.119,A -85,B 0,C 180,E1 -31113.27,E2 -31113.27} C_VEL
LIN {X 0,Y 36.237,Z 540.88,A -85,B 0,C 180,E1 -31125.861,E2 -31125.861} C_VEL
LIN {X 0,Y 49.667,Z 537.139,A -85,B 0,C 180,E1 -31132.095,E2 -31132.095} C_VEL
LIN {X 0,Y 59.979,Z 533.226,A -85,B 0,C 180,E1 -31134.858,E2 -31134.858} C_VEL
LIN {X 0,Y 70.392,Z 528.308,A -85,B 0,C 180,E1 -31136.76,E2 -31136.76} C_VEL
LIN {X 0,Y 80.863,Z 522.25,A -85,B 0,C 180,E1 -31138.154,E2 -31138.154} C_VEL
LIN {X 0,Y 91.372,Z 514.854,A -85,B 0,C 180,E1 -31139.184,E2 -31139.184} C_VEL
LIN {X 0,Y 101.905,Z 505.833,A -85,B 0,C 180,E1 -31140.092,E2 -31140.092} C_VEL
LIN {X 0,Y 105.421,Z 502.374,A -85,B 0,C 180,E1 -31140.366,E2 -31140.366} C_VEL
LIN {X 0,Y 105.424,Z 502.367,A -85,B 0,C 180,E1 -31140.598,E2 -31140.598} C_VEL
LIN {X 0,Y 94.905,Z 512.004,A -85,B 0,C 180,E1 -31141.404,E2 -31141.404} C_VEL
LIN {X 0,Y 84.414,Z 519.863,A -85,B 0,C 180,E1 -31142.489,E2 -31142.489} C_VEL
LIN {X 0,Y 76.559,Z 524.778,A -85,B 0,C 180,E1 -31143.458,E2 -31143.458} C_VEL
LIN {X 0,Y 69.9,Z 528.433,A -85,B 0,C 180,E1 -31143.946,E2 -31143.946} C_VEL
LIN {X 0,Y 58.333,Z 533.645,A -85,B 0,C 180,E1 -31143.351,E2 -31143.351} C_VEL
LIN {X 0,Y 48.784,Z 537.07,A -85,B 0,C 180,E1 -31142.556,E2 -31142.556} C_VEL
LIN {X 0,Y 41.485,Z 539.154,A -85,B 0,C 180,E1 -31142.784,E2 -31142.784} C_VEL
LIN {X 0,Y 39.048,Z 539.707,A -85,B 0,C 180,E1 -31143.252,E2 -31143.252} C_VEL
LIN {X 0,Y 28.317,Z 541.848,A -85,B 0,C 180,E1 -31146.899,E2 -31146.899} C_VEL
LIN {X 0,Y 14.905,Z 543.257,A -85,B 0,C 180,E1 -31159.432,E2 -31159.432} C_VEL
LIN {X 0,Y 8.941,Z 543.418,A -85,B 0,C 180,E1 -31178.178,E2 -31178.178} C_VEL
LIN {X 0,Y 5.923,Z 543.207,A -85,B 0,C 180,E1 -31229.996,E2 -31229.996} C_VEL
LIN {X 0,Y 9.303,Z 542.642,A -85,B 0,C 180,E1 -31279.062,E2 -31279.062} C_VEL
LIN {X 0,Y 21.826,Z 540.455,A -85,B 0,C 180,E1 -31305.01,E2 -31305.01} C_VEL
LIN {X 0,Y 35.478,Z 536.781,A -85,B 0,C 180,E1 -31312.077,E2 -31312.077} C_VEL
LIN {X 0,Y 46.561,Z 532.632,A -85,B 0,C 180,E1 -31314.85,E2 -31314.85} C_VEL
LIN {X 0,Y 56.331,Z 528.029,A -85,B 0,C 180,E1 -31316.44,E2 -31316.44} C_VEL
LIN {X 0,Y 63.32,Z 524.17,A -85,B 0,C 180,E1 -31317.317,E2 -31317.317} C_VEL
LIN {X 0,Y 63.31,Z 524.178,A -85,B 0,C 180,E1 -31317.513,E2 -31317.513} C_VEL
LIN {X 0,Y 52.722,Z 529.896,A -85,B 0,C 180,E1 -31318.731,E2 -31318.731} C_VEL
LIN {X 0,Y 42.169,Z 534.498,A -85,B 0,C 180,E1 -31320.622,E2 -31320.622} C_VEL
LIN {X 0,Y 31.691,Z 538.075,A -85,B 0,C 180,E1 -31323.707,E2 -31323.707} C_VEL
LIN {X 0,Y 21.355,Z 540.741,A -85,B 0,C 180,E1 -31329.155,E2 -31329.155} C_VEL
LIN {X 0,Y 8.693,Z 542.978,A -85,B 0,C 180,E1 -31356.062,E2 -31356.062} C_VEL
LIN {X 0,Y 5.725,Z 543.547,A -85,B 0,C 180,E1 -31410.004,E2 -31410.004} C_VEL
LIN {X 0,Y 8.717,Z 543.718,A -85,B 0,C 180,E1 -31463.73,E2 -31463.73} C_VEL
LIN {X 0,Y 21.367,Z 542.932,A -85,B 0,C 180,E1 -31490.66,E2 -31490.66} C_VEL
LIN {X 0,Y 35.18,Z 540.704,A -85,B 0,C 180,E1 -31497.249,E2 -31497.249} C_VEL
LIN {X 0,Y 49.196,Z 536.974,A -85,B 0,C 180,E1 -31500.37,E2 -31500.37} C_VEL
LIN {X 0,Y 49.205,Z 536.959,A -85,B 0,C 180,E1 -31501.137,E2 -31501.137} C_VEL
LIN {X 0,Y 39.048,Z 539.707,A -85,B 0,C 180,E1 -31503.252,E2 -31503.252} C_VEL
LIN {X 0,Y 37.52,Z 541.657,A -85,B 0,C 180,E1 -31503.653,E2 -31503.653} C_VEL
LIN {X 0,Y 37.52,Z 600,A -85,B 0,C 180,E1 -31503.653,E2 -31503.653} C_VEL
LIN {X 0,Y 37.52,Z 600,A -85,B 0,C 180,E1 -31503.653,E2 -31503.653}

QRS_NEXT_CUT()

QRS_NEXT()
QRS_HOME()

END
